// TIA Portal project "e199001v010" (V13)

(* hardware
DEVICE "Panel de operador_1"  KP900 Comfort
   slot 0: "HMI"  HMI  6AV2 124-1JC01-0AX0  13.0.1.0
   slot 1: "HMI_RT_1"  KP900 Comfort  6AV2 124-1JC01-0AX0  13.0.1.0
   slot 5: "Panel de operador_1.IE_CP_1"  Interfaz PROFINET
      slot 1: "Interfaz PROFINET_1"  Interfaz PROFINET
         slot 1: "Port_1"  Port
         slot 2: "Port_2"  Port
   slot 7: "Panel de operador_1.MPI/DP_CP_1"  Interfaz MPI/DP
*)

(* ===== HMI "HMI_RT_1" =====
connection "315_2DP": IF1 B, SIMATIC S7 300/400 MPI

HMI tags "Tabla de variables estándar"
   "Attendere1" : Byte, 1 s
   "LaserX" : Real, 1 s
   "TimeHBl" : S5Time, 1 s
   "SvoBobMin4" : Int, 1 s
   "PTMUX_MUXVAR_49" : Int, internal
   "Diam_filo10" : Real, 1 s
   "Color07" : Byte, 1 s
   "S_Int_1" : Int, 1 s
   "A_S_on07" : Bool, 1 s
   "TotalBlocks" : Int, 1 s
   "Diam_filo11" : Real, 1 s
   "Passo15" : Byte, 1 s
   "P14_Torque" : Int, 1 s
   "Trasf_Tipe" : Int, 1 s
   "DiamOutSvo" : Real, 1 s
   "CoefMul02" : Real, 1 s
   "PSvo_Current" : Int, 1 s
   "VelCin11" : Int, 1 s
   "R_F_Cur16" : Int, 1 s
   "P09_Power" : Int, 1 s
   "Q_elev" : Int, 1 s
   "RampJogDw" : Int, 1 s
   "RidMin14" : Int, 1 s
   "R_F_On07" : Bool, 1 s
   "TimLeft" : Real, 1 s
   "PTMUX_MUXVAR_45" : Int, internal
   "Q_bob_2" : Int, 1 s
   "P08_TempDriv" : Int, 1 s
   "VelMinChief" : Int, 1 s
   "P02_Speed" : Int, 1 s
   "Color05" : Byte, 1 s
   "Diam_filo14" : Real, 1 s
   "R_F_Cur01" : Int, 1 s
   "CoefMul03" : Real, 1 s
   "Mem_Rall" : Bool, 1 s
   "WearDieDw09" : Real, 1 s
   "P05_Current" : Int, 1 s
   "PTMUX_MUXVAR_46" : Int, internal
   "PTMUX_MUXVAR_37" : Int, internal
   "P07_Current" : Int, 1 s
   "R_F_On14" : Bool, 1 s
   "P06_Speed" : Int, 1 s
   "kW" : DInt, 1 s
   "Perc_WearAll" : Real, 1 s
   "Rall_manual" : Real, 1 s
   "SBPM_AGV_05" : Int, 1 s
   "Diam_filo04" : Real, 1 s
   "Ridu_12" : Int, 1 s
   "WearDieUp04" : Real, 1 s
   "WearDieDw14" : Real, 1 s
   "R_F_Cur06" : Int, 1 s
   "PTMUX_MUXVAR_10" : Int, internal
   "Check01" : Bool, 1 s
   "Gear5Elapsed" : Int, 1 s
   "Rst2" : Bool, 1 s
   "WearDieDw03" : Real, 1 s
   "AlTemQuad" : Int, 1 s
   "PJogL" : Int, 1 s
   "Diam_filo05" : Real, 1 s
   "RidMin10" : Int, 1 s
   "Color01" : Byte, 1 s
   "LaserOval" : Real, 1 s
   "PTMUX_MUXVAR_51" : Int, internal
   "RosetStat" : Byte, 1 s
   "WearDieDw04" : Real, 1 s
   "WearDieDw05" : Real, 1 s
   "P01_Speed" : Int, 1 s
   "P09_Current" : Int, 1 s
   "SBPM_AGV_12" : Int, 1 s
   "P05_Speed" : Int, 1 s
   "PBob_Power" : Int, 1 s
   "A_S_on05" : Bool, 1 s
   "Fil_rot_08" : Bool, 1 s
   "WearDieUp05" : Real, 1 s
   "Diam_filo02" : Real, 1 s
   "Passo11" : Byte, 1 s
   "PS_TempDrive" : Int, 1 s
   "P12_Torque" : Int, 1 s
   "Passo14" : Byte, 1 s
   "OTO_Actual" : Int, 1 s
   "Diam_Out" : Real, 1 s
   "Color09" : Byte, 1 s
   "OTO_Bargraph" : Int, 1 s
   "R_F_On15" : Bool, 1 s
   "P16_Current" : Int, 1 s
   "PTMUX_MUXVAR_26" : Int, internal
   "RidMin13" : Int, 1 s
   "Nr_recipe" : Int, 1 s
   "R_F_Cur15" : Int, 1 s
   "PTMUX_MUXVAR_53" : Int, internal
   "P13_Torque" : Int, 1 s
   "P12_Current" : Int, 1 s
   "PMat_Power" : Int, 1 s
   "P13_Current" : Int, 1 s
   "Matass" : Byte, 1 s
   "P16_Torque" : Int, 1 s
   "SvoBobMin2" : Int, 1 s
   "Color12" : Byte, 1 s
   "Fil_rot_01" : Bool, 1 s
   "PosizCarrell" : DInt, internal
   "SBPM_AGV_10" : Int, 1 s
   "BobMax1" : Int, 1 s
   "P15_Speed" : Int, 1 s
   "Ridu_06" : Int, 1 s
   "R_F_On10" : Bool, 1 s
   "WearDieUp09" : Real, 1 s
   "Acc_level" : Bool, 1 s
   "SvoBobMax1" : Int, 1 s
   "Diam_filo13" : Real, 1 s
   "D_Filt_Enc" : Int, 1 s
   "RidMin06" : Int, 1 s
   "Mux" : Int, 1 s
   "Fil_rot_09" : Bool, 1 s
   "PTMUX_MUXVAR_29" : Int, internal
   "VelMaxChief" : Int, 1 s
   "R_F_Cur14" : Int, 1 s
   "RidMin04" : Int, 1 s
   "SvoMax" : Int, 1 s
   "Counter_mat" : Real, 1 s
   "P15_Torque" : Int, 1 s
   "RidMin08" : Int, 1 s
   "PTMUX_MUXVAR_33" : Int, internal
   "CoefMul16" : Real, 1 s
   "P04_TempMot" : Int, 1 s
   "OTO_Min" : Int, 1 s
   "CoefMul09" : Real, 1 s
   "Gear4Elapsed" : Int, 1 s
   "P07_TempMot" : Int, 1 s
   "Ksensor" : Int, 1 s
   "CompAuto" : Bool, internal
   "Passo05" : Byte, 1 s
   "A_S_on01" : Bool, 1 s
   "P01_Torque" : Int, 1 s
   "Index" : Byte, 1 s
   "Tot_choic" : Byte, 1 s
   "WearDieUp12" : Real, 1 s
   "Fil_rot_10" : Bool, 1 s
   "Ridu_02" : Int, 1 s
   "Color08" : Byte, 1 s
   "RappDiam" : Int, 1 s   // E' il rapporto diametri bobine bobinatore
   "ControlSvo" : Bool, 1 s
   "DiamInSvo" : Real, 1 s
   "ControlStrat" : Bool, 1 s
   "Passo10" : Byte, 1 s
   "Laser2Thres" : Real, 1 s
   "SvoDiametro" : Int, 1 s
   "PTMUX_MUXVAR_25" : Int, internal
   "R_F_On03" : Bool, 1 s
   "Real_count" : Real, 1 s   // Metri parziali (prodotti)
   "Par_Type" : Byte, 1 s
   "TimeAccumulo" : Int, 1 s
   "P01_TempDriv" : Int, 1 s
   "Diam_filo06" : Real, 1 s
   "PSvo_Torque" : Int, 1 s
   "P10_Power" : Int, 1 s
   "VelCin14" : Int, 1 s
   "R_F_Cur12" : Int, 1 s
   "P15_Power" : Int, 1 s
   "Z_TIME" : WString[8], internal
   "GainCorr" : Int, 1 s
   "Diam_filo16" : Real, 1 s
   "RidMin16" : Int, 1 s
   "Pass_OTO" : Bool, 1 s   // Dichiarazione passo 1 se normale o OTO
   "CoefMul15" : Real, 1 s
   "PTMUX_MUXVAR_6" : Int, internal
   "Posizionam" : Int, internal
   "P03_TempMot" : Int, 1 s
   "WearDieDw02" : Real, 1 s
   "SBPM_AGV_04" : Int, 1 s
   "Passo06" : Byte, 1 s
   "PTMUX_MUXVAR_52" : Int, internal
   "P11_TempMot" : Int, 1 s
   "PTMUX_MUXVAR_1" : Int, internal
   "Elev_aut" : Bool, 1 s
   "Ridu_07" : Int, 1 s
   "Fil_rot_12" : Bool, 1 s
   "PTMUX_MUXVAR_7" : Int, internal
   "Param_Nr" : Int, 1 s
   "Passo02" : Byte, 1 s
   "VelCin08" : Int, 1 s
   "SBPM_AGV_15" : Int, 1 s
   "BobMin1" : Int, 1 s
   "Gear2Elapsed" : Int, 1 s
   "R_F_On02" : Bool, 1 s
   "Gear3Elapsed" : Int, 1 s
   "Diam_filo09" : Real, 1 s
   "P08_Speed" : Int, 1 s
   "R_F_On06" : Bool, 1 s
   "WearDieUp03" : Real, 1 s
   "SvoBobMin5" : Int, 1 s
   "SBPM_AGV_09" : Int, 1 s
   "Diam_filo03" : Real, 1 s
   "PTMUX_MUXVAR_8" : Int, internal
   "PTMUX_MUXVAR_16" : Int, internal
   "P13_Power" : Int, 1 s
   "Ridu_08" : Int, 1 s
   "PB_TempMot" : Int, 1 s
   "PTMUX_MUXVAR_27" : Int, internal
   "PT_Alarmas  1" : Array [0..19] of Int, 1 s
   "P07_Speed" : Int, 1 s
   "CoefMul10" : Real, 1 s
   "P11_TempDriv" : Int, 1 s
   "CoefMul07" : Real, 1 s
   "P13_TempMot" : Int, 1 s
   "Sfilaggio" : Bool, 1 s
   "P15_TempMot" : Int, 1 s
   "PTMUX_MUXVAR_36" : Int, internal
   "SBPM_AGV_16" : Int, 1 s
   "Ridu_16" : Int, 1 s
   "WearDieDw10" : Real, 1 s
   "VelCin06" : Int, 1 s
   "Gear4Set" : Int, 1 s
   "PMat_Torque" : Int, 1 s
   "VelCin03" : Int, 1 s
   "R_F_On11" : Bool, 1 s
   "DiamArrSvo" : Int, 1 s
   "Spool_choice" : Byte, 1 s
   "AGV_Set" : Bool, 1 s
   "R_F_Cur02" : Int, 1 s
   "CoefCorr" : Int, internal
   "WearDieUp14" : Real, 1 s
   "R_F_Cur08" : Int, 1 s
   "PMat_Speed" : Int, 1 s
   "LaserAlCh" : Bool, 1 s
   "PTMUX_MUXVAR_54" : Int, internal
   "Ridu_14" : Int, 1 s
   "Allineam" : Bool, 1 s
   "WearDieDw01" : Real, 1 s
   "Color04" : Byte, 1 s
   "Counter_traf" : Real, 1 s
   "PMat_Current" : Int, 1 s
   "PTMUX_MUXVAR_50" : Int, internal
   "OffAnalIn" : Int, 1 s
   "A_S_on16" : Bool, 1 s
   "PBobin" : Byte, 1 s
   "Diam_filo12" : Real, 1 s
   "VelMat" : Int, 1 s
   "PTMUX_MUXVAR_40" : Int, internal
   "PTMUX_MUXVAR_31" : Int, internal
   "SvoBobMax6" : Int, 1 s
   "Passo07" : Byte, 1 s
   "P09_TempDriv" : Int, 1 s
   "Pes_Specif" : Real, 1 s
   "Passo01" : Byte, 1 s
   "Ridu_01" : Int, 1 s
   "RappStrat3" : Int, 1 s
   "Fil_rot_05" : Bool, 1 s
   "P05_TempMot" : Int, 1 s
   "WearDieUp06" : Real, 1 s
   "WearDieUp11" : Real, 1 s
   "VelCin09" : Int, 1 s
   "P04_Torque" : Int, 1 s
   "P15_TempDriv" : Int, 1 s
   "PTMUX_MUXVAR_17" : Int, internal
   "Sirena" : Bool, 1 s
   "Perc_WearAvv" : Real, 1 s
   "PTMUX_MUXVAR_5" : Int, internal
   "PTMUX_MUXVAR_39" : Int, internal
   "PT_Acuses OP  2" : Array [0..4] of Word, 1 s
   "PTMUX_MUXVAR_47" : Int, internal
   "PTMUX_MUXVAR_24" : Int, internal
   "kg_total" : Real, 1 s
   "Gear5Set" : Int, 1 s
   "P07_Power" : Int, 1 s
   "JogDestra" : Int, internal
   "PTMUX_MUXVAR_38" : Int, internal
   "VelCin13" : Int, 1 s
   "P07_TempDriv" : Int, 1 s
   "Check05" : Bool, 1 s
   "P14_Power" : Int, 1 s
   "Ridu_10" : Int, 1 s
   "P09_Speed" : Int, 1 s
   "Fil_rot_11" : Bool, 1 s
   "Color13" : Byte, 1 s
   "BobTipo" : Bool, 1 s
   "Color03" : Byte, 1 s
   "Q_bob_3" : Int, 1 s
   "TimeForche" : S5Time, 1 s
   "Gear1Elapsed" : Int, 1 s
   "Imp_Exp" : Bool, 1 s
   "VelCin01" : Int, 1 s
   "PM_TempMot" : Int, 1 s
   "Rst1" : Bool, 1 s
   "Total" : Real, 1 s
   "PSvo_Power" : Int, 1 s
   "R_F_Cur09" : Int, 1 s
   "Stato_Linea" : Int, 1 s   // Visualizzazione stato linea
   "Q_bob_5" : Int, 1 s
   "Passo08" : Byte, 1 s
   "Vel_impostat" : Int, 1 s
   "CoefMul06" : Real, 1 s
   "P09_Torque" : Int, 1 s
   "PS_TempMot" : Int, 1 s
   "Gear1Set" : Int, 1 s
   "PTMUX_MUXVAR_35" : Int, internal
   "Exp_ImpQuest" : Bool, 1 s
   "SvoBobMin6" : Int, 1 s
   "Ridu_13" : Int, 1 s
   "SBPM" : Bool, 1 s   // Dichiarazione passo 1 se normale o OTO
   "RicFlangia" : Int, internal
   "A_S_on03" : Bool, 1 s
   "RidMin01" : Int, 1 s
   "OTO_BarUP" : Int, 1 s
   "Check02" : Bool, 1 s
   "TimeH2Fil" : S5Time, 1 s
   "PT_Acuses OP  1" : Array [0..9] of Int, 1 s
   "P11_Torque" : Int, 1 s
   "P14_TempDriv" : Int, 1 s
   "Life_hours" : DInt, 1 s
   "Ral_Aut_Cal" : Real, 1 s
   "JogSinistra" : Int, internal
   "P10_TempDriv" : Int, 1 s
   "PTMUX_MUXVAR_32" : Int, internal
   "A_S_on06" : Bool, 1 s
   "CoefMul05" : Real, 1 s
   "P03_Torque" : Int, 1 s
   "Fil_rot_03" : Bool, 1 s
   "P15_Current" : Int, 1 s
   "A_S_on14" : Bool, 1 s
   "SvoBobMin1" : Int, 1 s
   "RappStrat2" : Int, 1 s
   "P08_TempMot" : Int, 1 s
   "P03_Speed" : Int, 1 s
   "PTMUX_MUXVAR_34" : Int, internal
   "PTMUX_MUXVAR_30" : Int, internal
   "P14_Speed" : Int, 1 s
   "A_S_on12" : Bool, 1 s
   "Imp_count" : Real, 1 s   // Metri impostati
   "P04_TempDriv" : Int, 1 s
   "R_F_On09" : Bool, 1 s
   "JogStrat" : Int, 1 s
   "RappStrat1" : Int, 1 s
   "A_S_on13" : Bool, 1 s
   "Color02" : Byte, 1 s
   "SvoMin" : Int, 1 s
   "VelCin12" : Int, 1 s
   "RappStrat4" : Int, 1 s
   "K_Stratific" : Int, 1 s
   "BobMax2" : Int, 1 s
   "RidMin02" : Int, 1 s
   "P06_TempMot" : Int, 1 s
   "P05_Torque" : Int, 1 s
   "RidMin05" : Int, 1 s
   "SvoBobMax4" : Int, 1 s
   "OTO_MinRid" : Int, 1 s
   "Passo09" : Byte, 1 s
   "P02_Torque" : Int, 1 s
   "SistMisure" : Bool, 1 s
   "RosettVel" : Int, 1 s
   "PTMUX_MUXVAR_12" : Int, internal
   "BobCoppia" : Int, 1 s
   "SBPM_AGV_11" : Int, 1 s
   "CoefMul12" : Real, 1 s
   "PTMUX_MUXVAR_19" : Int, internal
   "Diam_filo01" : Real, 1 s
   "S_Int_5" : Int, 1 s
   "P02_Current" : Int, 1 s
   "MaxSens" : Int, 1 s
   "Block_Choice" : Int, 1 s
   "P10_Speed" : Int, 1 s
   "RidMin12" : Int, 1 s
   "R_F_Cur03" : Int, 1 s
   "R_F_Cur07" : Int, 1 s
   "PTMUX_MUXVAR_56" : Int, internal
   "Domanda" : Bool, 1 s
   "S_IntTime" : Int, 1 s
   "PTMUX_MUXVAR_41" : Int, internal
   "Ridu_09" : Int, 1 s
   "VelCin15" : Int, 1 s
   "A_S_on02" : Bool, 1 s
   "Ridu_11" : Int, 1 s
   "P16_Speed" : Int, 1 s
   "CoefMul04" : Real, 1 s
   "PTMUX_MUXVAR_2" : Int, internal
   "P07_Torque" : Int, 1 s
   "Color11" : Byte, 1 s
   "P04_Current" : Int, 1 s
   "Passo04" : Byte, 1 s
   "LaserY" : Real, 1 s
   "LaserMedio" : Real, 1 s
   "kg" : Bool, internal
   "WearDieUp01" : Real, 1 s
   "R_F_Cur05" : Int, 1 s
   "Ridu_15" : Int, 1 s
   "Diam_filo08" : Real, 1 s
   "P12_Speed" : Int, 1 s
   "Contametri" : Byte, 1 s
   "PBob_Speed" : Int, 1 s
   "WearDieUp07" : Real, 1 s
   "SBPM_AGV_03" : Int, 1 s
   "VelCin02" : Int, 1 s
   "RidMin11" : Int, 1 s
   "BobMin2" : Int, 1 s
   "Sens_Gain" : Int, 1 s
   "PTMUX_MUXVAR_22" : Int, internal
   "Color14" : Byte, 1 s
   "A_S_on11" : Bool, 1 s
   "InvSinistra" : Int, internal
   "P08_Torque" : Int, 1 s
   "PTMUX_MUXVAR_57" : Int, internal
   "Rst4" : Bool, 1 s
   "R_F_Cur10" : Int, 1 s
   "Color16" : Byte, 1 s
   "PBob_Torque" : Int, 1 s
   "PTMUX_MUXVAR_23" : Int, internal
   "P08_Current" : Int, 1 s
   "PTMUX_MUXVAR_11" : Int, internal
   "P02_TempMot" : Int, 1 s
   "Svolgitore" : Byte, 1 s
   "Gear2Set" : Int, 1 s
   "P02_TempDriv" : Int, 1 s
   "SBPM_AGV_07" : Int, 1 s
   "Elevator" : Bool, 1 s
   "A_S_on10" : Bool, 1 s
   "VelCin10" : Int, 1 s
   "PT_Alarmas  2" : Array [0..9] of Word, 1 s
   "CoefMul11" : Real, 1 s
   "Color10" : Byte, 1 s
   "Rst3" : Bool, 1 s
   "P03_Power" : Int, 1 s
   "R_F_On08" : Bool, 1 s
   "SvoBobMax3" : Int, 1 s
   "P10_TempMot" : Int, 1 s
   "PTMUX_MUXVAR_44" : Int, internal
   "WearDieUp10" : Real, 1 s
   "PAct_Sen" : Int, 1 s
   "Sel_count" : Bool, 1 s
   "Diam_filo07" : Real, 1 s
   "R_F_On13" : Bool, 1 s
   "Fil_rot_06" : Bool, 1 s
   "PTMUX_MUXVAR_43" : Int, internal
   "CoefMul14" : Real, 1 s
   "Fil_rot_04" : Bool, 1 s
   "Fast_Dw" : Int, 1 s
   "PTMUX_MUXVAR_20" : Int, internal
   "PTMUX_MUXVAR_15" : Int, internal
   "Svo_Spools" : Byte, 1 s
   "SvoBobMax2" : Int, 1 s
   "kg_parz" : Real, 1 s
   "Attendere" : Bool, 1 s
   "R_F_Cur04" : Int, 1 s
   "AGV" : DInt, 1 s
   "T_Rosett" : Int, internal
   "R_F_Cur13" : Int, 1 s
   "P04_Speed" : Int, 1 s
   "PJogV" : Int, 1 s
   "Fil_rot_07" : Bool, 1 s
   "BobTirVel" : Bool, 1 s
   "S_Rosett" : Int, internal
   "PTMUX_MUXVAR_14" : Int, internal
   "VelCin16" : Int, 1 s
   "PTMUX_MUXVAR_18" : Int, internal
   "Ridu_04" : Int, 1 s
   "Real_Sens" : Int, 1 s
   "PTMUX_MUXVAR_55" : Int, internal
   "Color06" : Byte, 1 s
   "Q_bob_6" : Int, 1 s
   "OTOMotorized" : Bool, 1 s   // Dichiarazione passo 1 motorizzato o no
   "RidMin07" : Int, 1 s
   "Passo16" : Byte, 1 s
   "Gear3Set" : Int, 1 s
   "RampJogUp" : Int, 1 s
   "WearDieDw07" : Real, 1 s
   "P06_Current" : Int, 1 s
   "SvoBobMin3" : Int, 1 s
   "PTMUX_MUXVAR_28" : Int, internal
   "Diam_filoM" : Real, 1 s
   "Passo12" : Byte, 1 s
   "SBPM_AGV_01" : Int, 1 s
   "WearDieUp13" : Real, 1 s
   "Rosett" : Bool, 1 s
   "Fil_rot_14" : Bool, 1 s
   "Attendere3" : Byte, 1 s
   "WearDieDw06" : Real, 1 s
   "R_F_On16" : Bool, 1 s
   "P16_TempMot" : Int, 1 s
   "WearDieDw12" : Real, 1 s
   "Passo13" : Byte, 1 s
   "RidMin03" : Int, 1 s
   "PTMUX_MUXVAR_9" : Int, internal
   "Diam_filo15" : Real, 1 s
   "P08_Power" : Int, 1 s
   "LaserChoic" : Bool, 1 s
   "P16_Power" : Int, 1 s
   "OTO_Imposed" : Int, 1 s
   "WearDieUp08" : Real, 1 s
   "DiamManual" : Real, 1 s
   "A_S_on09" : Bool, 1 s
   "PT_Imagen de los LED  1" : Array [0..3] of Int, 1 s
   "CoefMul01" : Real, 1 s
   "P09_TempMot" : Int, 1 s
   "Check03" : Bool, 1 s
   "Task_Id" : Int, 1 s
   "OTO_Rid" : Int, 1 s
   "P02_Power" : Int, 1 s
   "DistanzaPx" : DInt, internal
   "LaserStato" : Int, 1 s
   "Recipe_Wait" : Int, 1 s
   "OutChoice" : Byte, 1 s
   "A_S_on08" : Bool, 1 s
   "P06_Power" : Int, 1 s
   "Ridu_03" : Int, 1 s
   "TempQuad" : Int, 1 s
   "R_F_On01" : Bool, 1 s
   "PTMUX_MUXVAR_42" : Int, internal
   "P11_Current" : Int, 1 s
   "PTMUX_MUXVAR_3" : Int, internal
   "S_Int_4" : Int, 1 s
   "VelRal" : Int, 1 s
   "R_F_Cur11" : Int, 1 s
   "Color15" : Byte, 1 s
   "Worked_hours" : DInt, 1 s
   "OTO_Max" : Int, 1 s
   "P06_Torque" : Int, 1 s
   "kg_imp" : Real, 1 s
   "A_S_on04" : Bool, 1 s
   "AnticipoSvo" : Int, 1 s
   "D_Prop_1" : Int, 1 s
   "VelSfilag" : Int, 1 s
   "Slow_Up" : Int, 1 s
   "R_F_On12" : Bool, 1 s
   "PTMUX_MUXVAR_13" : Int, internal
   "Fil_rot_16" : Bool, 1 s
   "P04_Power" : Int, 1 s
   "PTMUX_MUXVAR_4" : Int, internal
   "SBPM_AGV_14" : Int, 1 s
   "RealSpINT" : Int, 1 s   // Velocita' m/s in REAL
   "WearDieUp02" : Real, 1 s
   "P03_Current" : Int, 1 s
   "WearDieDw11" : Real, 1 s
   "P10_Torque" : Int, 1 s
   "WearDieDw08" : Real, 1 s
   "OTO_BarDW" : Int, 1 s
   "P12_TempDriv" : Int, 1 s
   "R_F_On05" : Bool, 1 s
   "Rst5" : Bool, 1 s
   "VelCin07" : Int, 1 s
   "Attesa2" : Bool, 1 s
   "PSvo_Speed" : Int, 1 s
   "P14_Current" : Int, 1 s
   "S_Int_2" : Int, 1 s
   "S_Prop_2" : Int, 1 s
   "P12_Power" : Int, 1 s
   "Passo03" : Byte, 1 s
   "P13_TempDriv" : Int, 1 s
   "Laser1Thres" : Real, 1 s
   "Attesa1" : Bool, 1 s
   "CoefMul13" : Real, 1 s
   "Fil_rot_15" : Bool, 1 s
   "P01_Power" : Int, 1 s
   "SBPM_AGV_02" : Int, 1 s
   "D_Int" : Int, 1 s
   "Z_DATE" : WString[10], internal
   "CoefMul08" : Real, 1 s
   "Check04" : Bool, 1 s
   "PTMUX_MUXVAR_21" : Int, internal
   "P12_TempMot" : Int, 1 s
   "ON_SS" : Byte, 1 s
   "SBPM_AGV_13" : Int, 1 s
   "P10_Current" : Int, 1 s
   "MinSens" : Int, 1 s
   "Q_bob_1" : Int, 1 s
   "Slow_dw" : Int, 1 s
   "Max_vel" : Int, 1 s
   "SBPM_AGV_08" : Int, 1 s
   "S_Prop_1" : Int, 1 s
   "Fil_rot_13" : Bool, 1 s
   "BypassDati" : Bool, 1 s
   "PM_TempDriv" : Int, 1 s
   "P13_Speed" : Int, 1 s
   "Reset_kW" : Bool, 1 s
   "P01_Current" : Int, 1 s
   "A_S_on15" : Bool, 1 s
   "PB_TempDrive" : Int, 1 s
   "Q_bob_4" : Int, 1 s
   "BobTiro" : Int, 1 s
   "TimeVenBloc" : S5Time, 1 s
   "PTMUX_MUXVAR_48" : Int, internal
   "P11_Power" : Int, 1 s
   "Die_Wear_Ch" : Byte, 1 s
   "D_Prop_2" : Int, 1 s
   "P16_TempDriv" : Int, 1 s
   "WearDieDw13" : Real, 1 s
   "Value" : DInt, 1 s
   "SvoBobMax5" : Int, 1 s
   "RidMin15" : Int, 1 s
   "ColorSvolg" : Byte, 1 s
   "Ridu_05" : Int, 1 s
   "PT_Avisos de servicio  1" : Array [0..4] of Int, 1 s
   "R_F_On04" : Bool, 1 s
   "P03_TempDriv" : Int, 1 s
   "VelCin05" : Int, 1 s
   "P11_Speed" : Int, 1 s
   "SBPM_AGV_06" : Int, 1 s
   "Mux1" : Int, 1 s
   "VelCin04" : Int, 1 s
   "PBob_Current" : Int, 1 s
   "InvDestra" : Int, internal
   "P14_TempMot" : Int, 1 s
   "P06_TempDriv" : Int, 1 s
   "P01_TempMot" : Int, 1 s
   "Min_vel" : Int, 1 s
   "P05_TempDriv" : Int, 1 s
   "TimeStratCal" : Int, 1 s
   "P05_Power" : Int, 1 s
   "BobDiametro" : Int, 1 s
   "Sens_Deriv" : Int, 1 s
   "Pilota" : Int, 1 s
   "Fil_rot_02" : Bool, 1 s
   "Time_1" : DateTime, internal

discrete alarms
   43: '', class Warnings, trigger "PT_Avisos de servicio  1" bit 42
   2018: '', class Errors, trigger "PT_Acuses OP  1" bit 17
   2209: '', class Errors, trigger "PT_Acuses OP  2" bit 48
   2034: '', class Errors, trigger "PT_Acuses OP  1" bit 33
   17: '', class Warnings, trigger "PT_Avisos de servicio  1" bit 16
   2: '', class Warnings, trigger "PT_Avisos de servicio  1" bit 1
   2189: '', class Errors, trigger "PT_Acuses OP  2" bit 28
   2129: '', class Errors, trigger "PT_Acuses OP  1" bit 128
   2019: '', class Errors, trigger "PT_Acuses OP  1" bit 18
   2098: '', class Errors, trigger "PT_Acuses OP  1" bit 97
   2072: '', class Errors, trigger "PT_Acuses OP  1" bit 71
   24: '', class Warnings, trigger "PT_Avisos de servicio  1" bit 23
   2188: '', class Errors, trigger "PT_Acuses OP  2" bit 27
   2181: '', class Errors, trigger "PT_Acuses OP  2" bit 20
   2014: '', class Errors, trigger "PT_Acuses OP  1" bit 13
   2049: '', class Errors, trigger "PT_Acuses OP  1" bit 48
   2141: '', class Errors, trigger "PT_Acuses OP  1" bit 140
   10: '', class Warnings, trigger "PT_Avisos de servicio  1" bit 9
   2023: '', class Errors, trigger "PT_Acuses OP  1" bit 22
   2031: '', class Errors, trigger "PT_Acuses OP  1" bit 30
   2219: '', class Errors, trigger "PT_Acuses OP  2" bit 58
   2200: '', class Errors, trigger "PT_Acuses OP  2" bit 39
   40: '', class Warnings, trigger "PT_Avisos de servicio  1" bit 39
   2193: '', class Errors, trigger "PT_Acuses OP  2" bit 32
   2128: '', class Errors, trigger "PT_Acuses OP  1" bit 127
   2140: '', class Errors, trigger "PT_Acuses OP  1" bit 139
   2053: '', class Errors, trigger "PT_Acuses OP  1" bit 52
   70: '', class Warnings, trigger "PT_Avisos de servicio  1" bit 69
   2061: '', class Errors, trigger "PT_Acuses OP  1" bit 60
   2135: '', class Errors, trigger "PT_Acuses OP  1" bit 134
   2126: '', class Errors, trigger "PT_Acuses OP  1" bit 125
   2065: '', class Errors, trigger "PT_Acuses OP  1" bit 64
   2206: '', class Errors, trigger "PT_Acuses OP  2" bit 45
   73: '', class Warnings, trigger "PT_Avisos de servicio  1" bit 72
   2199: '', class Errors, trigger "PT_Acuses OP  2" bit 38
   71: '', class Warnings, trigger "PT_Avisos de servicio  1" bit 70
   2158: '', class Errors, trigger "PT_Acuses OP  1" bit 157
   2038: '', class Errors, trigger "PT_Acuses OP  1" bit 37
   19: '', class Warnings, trigger "PT_Avisos de servicio  1" bit 18
   2081: '', class Errors, trigger "PT_Acuses OP  1" bit 80
   37: '', class Warnings, trigger "PT_Avisos de servicio  1" bit 36
   3: '', class Warnings, trigger "PT_Avisos de servicio  1" bit 2
   2238: '', class Errors, trigger "PT_Acuses OP  2" bit 77
   2201: '', class Errors, trigger "PT_Acuses OP  2" bit 40
   2008: '', class Errors, trigger "PT_Acuses OP  1" bit 7
   2032: '', class Errors, trigger "PT_Acuses OP  1" bit 31
   2145: '', class Errors, trigger "PT_Acuses OP  1" bit 144
   2143: '', class Errors, trigger "PT_Acuses OP  1" bit 142
   2134: '', class Errors, trigger "PT_Acuses OP  1" bit 133
   2056: '', class Errors, trigger "PT_Acuses OP  1" bit 55
   2004: '', class Errors, trigger "PT_Acuses OP  1" bit 3
   2043: '', class Errors, trigger "PT_Acuses OP  1" bit 42
   2216: '', class Errors, trigger "PT_Acuses OP  2" bit 55
   2234: '', class Errors, trigger "PT_Acuses OP  2" bit 73
   27: '', class Warnings, trigger "PT_Avisos de servicio  1" bit 26
   2133: '', class Errors, trigger "PT_Acuses OP  1" bit 132
   2113: '', class Errors, trigger "PT_Acuses OP  1" bit 112
   31: '', class Warnings, trigger "PT_Avisos de servicio  1" bit 30
   2170: '', class Errors, trigger "PT_Acuses OP  2" bit 9
   2162: '', class Errors, trigger "PT_Acuses OP  2" bit 1
   29: '', class Warnings, trigger "PT_Avisos de servicio  1" bit 28
   2187: '', class Errors, trigger "PT_Acuses OP  2" bit 26
   2094: '', class Errors, trigger "PT_Acuses OP  1" bit 93
   2041: '', class Errors, trigger "PT_Acuses OP  1" bit 40
   2076: '', class Errors, trigger "PT_Acuses OP  1" bit 75
   2084: '', class Errors, trigger "PT_Acuses OP  1" bit 83
   2215: '', class Errors, trigger "PT_Acuses OP  2" bit 54
   2131: '', class Errors, trigger "PT_Acuses OP  1" bit 130
   2195: '', class Errors, trigger "PT_Acuses OP  2" bit 34
   2205: '', class Errors, trigger "PT_Acuses OP  2" bit 44
   78: '', class Warnings, trigger "PT_Avisos de servicio  1" bit 77
   2079: '', class Errors, trigger "PT_Acuses OP  1" bit 78
   2068: '', class Errors, trigger "PT_Acuses OP  1" bit 67
   2196: '', class Errors, trigger "PT_Acuses OP  2" bit 35
   2123: '', class Errors, trigger "PT_Acuses OP  1" bit 122
   2152: '', class Errors, trigger "PT_Acuses OP  1" bit 151
   2112: '', class Errors, trigger "PT_Acuses OP  1" bit 111
   2211: '', class Errors, trigger "PT_Acuses OP  2" bit 50
   2077: '', class Errors, trigger "PT_Acuses OP  1" bit 76
   46: '', class Warnings, trigger "PT_Avisos de servicio  1" bit 45
   77: '', class Warnings, trigger "PT_Avisos de servicio  1" bit 76
   33: '', class Warnings, trigger "PT_Avisos de servicio  1" bit 32
   2148: '', class Errors, trigger "PT_Acuses OP  1" bit 147
   2064: '', class Errors, trigger "PT_Acuses OP  1" bit 63
   65: '', class Warnings, trigger "PT_Avisos de servicio  1" bit 64
   2237: '', class Errors, trigger "PT_Acuses OP  2" bit 76
   79: '', class Warnings, trigger "PT_Avisos de servicio  1" bit 78
   2218: '', class Errors, trigger "PT_Acuses OP  2" bit 57
   2075: '', class Errors, trigger "PT_Acuses OP  1" bit 74
   2167: '', class Errors, trigger "PT_Acuses OP  2" bit 6
   2073: '', class Errors, trigger "PT_Acuses OP  1" bit 72
   2225: '', class Errors, trigger "PT_Acuses OP  2" bit 64
   2070: '', class Errors, trigger "PT_Acuses OP  1" bit 69
   2222: '', class Errors, trigger "PT_Acuses OP  2" bit 61
   22: '', class Warnings, trigger "PT_Avisos de servicio  1" bit 21
   2092: '', class Errors, trigger "PT_Acuses OP  1" bit 91
   2208: '', class Errors, trigger "PT_Acuses OP  2" bit 47
   56: '', class Warnings, trigger "PT_Avisos de servicio  1" bit 55
   6: '', class Warnings, trigger "PT_Avisos de servicio  1" bit 5
   25: '', class Warnings, trigger "PT_Avisos de servicio  1" bit 24
   2045: '', class Errors, trigger "PT_Acuses OP  1" bit 44
   2161: '', class Errors, trigger "PT_Acuses OP  2" bit 0
   2122: '', class Errors, trigger "PT_Acuses OP  1" bit 121
   2192: '', class Errors, trigger "PT_Acuses OP  2" bit 31
   2108: '', class Errors, trigger "PT_Acuses OP  1" bit 107
   2011: '', class Errors, trigger "PT_Acuses OP  1" bit 10
   2230: '', class Errors, trigger "PT_Acuses OP  2" bit 69
   2052: '', class Errors, trigger "PT_Acuses OP  1" bit 51
   2163: '', class Errors, trigger "PT_Acuses OP  2" bit 2
   2027: '', class Errors, trigger "PT_Acuses OP  1" bit 26
   2093: '', class Errors, trigger "PT_Acuses OP  1" bit 92
   2026: '', class Errors, trigger "PT_Acuses OP  1" bit 25
   68: '', class Warnings, trigger "PT_Avisos de servicio  1" bit 67
   2144: '', class Errors, trigger "PT_Acuses OP  1" bit 143
   2150: '', class Errors, trigger "PT_Acuses OP  1" bit 149
   2005: '', class Errors, trigger "PT_Acuses OP  1" bit 4
   2036: '', class Errors, trigger "PT_Acuses OP  1" bit 35
   72: '', class Warnings, trigger "PT_Avisos de servicio  1" bit 71
   2040: '', class Errors, trigger "PT_Acuses OP  1" bit 39
   48: '', class Warnings, trigger "PT_Avisos de servicio  1" bit 47
   2146: '', class Errors, trigger "PT_Acuses OP  1" bit 145
   2042: '', class Errors, trigger "PT_Acuses OP  1" bit 41
   55: '', class Warnings, trigger "PT_Avisos de servicio  1" bit 54
   2174: '', class Errors, trigger "PT_Acuses OP  2" bit 13
   2210: '', class Errors, trigger "PT_Acuses OP  2" bit 49
   2235: '', class Errors, trigger "PT_Acuses OP  2" bit 74
   5: '', class Warnings, trigger "PT_Avisos de servicio  1" bit 4
   57: '', class Warnings, trigger "PT_Avisos de servicio  1" bit 56
   74: '', class Warnings, trigger "PT_Avisos de servicio  1" bit 73
   2137: '', class Errors, trigger "PT_Acuses OP  1" bit 136
   2138: '', class Errors, trigger "PT_Acuses OP  1" bit 137
   80: '', class Warnings, trigger "PT_Avisos de servicio  1" bit 79
   2062: '', class Errors, trigger "PT_Acuses OP  1" bit 61
   8: '', class Warnings, trigger "PT_Avisos de servicio  1" bit 7
   2178: '', class Errors, trigger "PT_Acuses OP  2" bit 17
   11: '', class Warnings, trigger "PT_Avisos de servicio  1" bit 10
   2217: '', class Errors, trigger "PT_Acuses OP  2" bit 56
   13: '', class Warnings, trigger "PT_Avisos de servicio  1" bit 12
   2149: '', class Errors, trigger "PT_Acuses OP  1" bit 148
   2120: '', class Errors, trigger "PT_Acuses OP  1" bit 119
   2213: '', class Errors, trigger "PT_Acuses OP  2" bit 52
   2207: '', class Errors, trigger "PT_Acuses OP  2" bit 46
   2071: '', class Errors, trigger "PT_Acuses OP  1" bit 70
   2033: '', class Errors, trigger "PT_Acuses OP  1" bit 32
   2059: '', class Errors, trigger "PT_Acuses OP  1" bit 58
   2088: '', class Errors, trigger "PT_Acuses OP  1" bit 87
   2010: '', class Errors, trigger "PT_Acuses OP  1" bit 9
   2156: '', class Errors, trigger "PT_Acuses OP  1" bit 155
   2022: '', class Errors, trigger "PT_Acuses OP  1" bit 21
   7: '', class Warnings, trigger "PT_Avisos de servicio  1" bit 6
   2047: '', class Errors, trigger "PT_Acuses OP  1" bit 46
   2090: '', class Errors, trigger "PT_Acuses OP  1" bit 89
   2074: '', class Errors, trigger "PT_Acuses OP  1" bit 73
   15: '', class Warnings, trigger "PT_Avisos de servicio  1" bit 14
   4: '', class Warnings, trigger "PT_Avisos de servicio  1" bit 3
   2025: '', class Errors, trigger "PT_Acuses OP  1" bit 24
   75: '', class Warnings, trigger "PT_Avisos de servicio  1" bit 74
   61: '', class Warnings, trigger "PT_Avisos de servicio  1" bit 60
   2114: '', class Errors, trigger "PT_Acuses OP  1" bit 113
   2091: '', class Errors, trigger "PT_Acuses OP  1" bit 90
   2117: '', class Errors, trigger "PT_Acuses OP  1" bit 116
   21: '', class Warnings, trigger "PT_Avisos de servicio  1" bit 20
   49: '', class Warnings, trigger "PT_Avisos de servicio  1" bit 48
   2153: '', class Errors, trigger "PT_Acuses OP  1" bit 152
   50: '', class Warnings, trigger "PT_Avisos de servicio  1" bit 49
   32: '', class Warnings, trigger "PT_Avisos de servicio  1" bit 31
   2030: '', class Errors, trigger "PT_Acuses OP  1" bit 29
   2085: '', class Errors, trigger "PT_Acuses OP  1" bit 84
   2116: '', class Errors, trigger "PT_Acuses OP  1" bit 115
   2173: '', class Errors, trigger "PT_Acuses OP  2" bit 12
   2194: '', class Errors, trigger "PT_Acuses OP  2" bit 33
   2080: '', class Errors, trigger "PT_Acuses OP  1" bit 79
   2009: '', class Errors, trigger "PT_Acuses OP  1" bit 8
   16: '', class Warnings, trigger "PT_Avisos de servicio  1" bit 15
   2055: '', class Errors, trigger "PT_Acuses OP  1" bit 54
   2078: '', class Errors, trigger "PT_Acuses OP  1" bit 77
   2159: '', class Errors, trigger "PT_Acuses OP  1" bit 158
   76: '', class Warnings, trigger "PT_Avisos de servicio  1" bit 75
   2171: '', class Errors, trigger "PT_Acuses OP  2" bit 10
   2233: '', class Errors, trigger "PT_Acuses OP  2" bit 72
   2035: '', class Errors, trigger "PT_Acuses OP  1" bit 34
   2104: '', class Errors, trigger "PT_Acuses OP  1" bit 103
   2226: '', class Errors, trigger "PT_Acuses OP  2" bit 65
   2186: '', class Errors, trigger "PT_Acuses OP  2" bit 25
   2115: '', class Errors, trigger "PT_Acuses OP  1" bit 114
   2125: '', class Errors, trigger "PT_Acuses OP  1" bit 124
   2050: '', class Errors, trigger "PT_Acuses OP  1" bit 49
   45: '', class Warnings, trigger "PT_Avisos de servicio  1" bit 44
   2157: '', class Errors, trigger "PT_Acuses OP  1" bit 156
   2086: '', class Errors, trigger "PT_Acuses OP  1" bit 85
   2087: '', class Errors, trigger "PT_Acuses OP  1" bit 86
   2111: '', class Errors, trigger "PT_Acuses OP  1" bit 110
   2183: '', class Errors, trigger "PT_Acuses OP  2" bit 22
   2180: '', class Errors, trigger "PT_Acuses OP  2" bit 19
   2166: '', class Errors, trigger "PT_Acuses OP  2" bit 5
   2048: '', class Errors, trigger "PT_Acuses OP  1" bit 47
   2142: '', class Errors, trigger "PT_Acuses OP  1" bit 141
   58: '', class Warnings, trigger "PT_Avisos de servicio  1" bit 57
   2101: '', class Errors, trigger "PT_Acuses OP  1" bit 100
   9: '', class Warnings, trigger "PT_Avisos de servicio  1" bit 8
   2185: '', class Errors, trigger "PT_Acuses OP  2" bit 24
   2229: '', class Errors, trigger "PT_Acuses OP  2" bit 68
   1: '', class Warnings, trigger "PT_Avisos de servicio  1" bit 0
   2154: '', class Errors, trigger "PT_Acuses OP  1" bit 153
   2082: '', class Errors, trigger "PT_Acuses OP  1" bit 81
   2124: '', class Errors, trigger "PT_Acuses OP  1" bit 123
   2103: '', class Errors, trigger "PT_Acuses OP  1" bit 102
   2169: '', class Errors, trigger "PT_Acuses OP  2" bit 8
   2236: '', class Errors, trigger "PT_Acuses OP  2" bit 75
   2164: '', class Errors, trigger "PT_Acuses OP  2" bit 3
   2118: '', class Errors, trigger "PT_Acuses OP  1" bit 117
   2106: '', class Errors, trigger "PT_Acuses OP  1" bit 105
   2139: '', class Errors, trigger "PT_Acuses OP  1" bit 138
   2202: '', class Errors, trigger "PT_Acuses OP  2" bit 41
   39: '', class Warnings, trigger "PT_Avisos de servicio  1" bit 38
   67: '', class Warnings, trigger "PT_Avisos de servicio  1" bit 66
   2107: '', class Errors, trigger "PT_Acuses OP  1" bit 106
   2231: '', class Errors, trigger "PT_Acuses OP  2" bit 70
   2024: '', class Errors, trigger "PT_Acuses OP  1" bit 23
   2177: '', class Errors, trigger "PT_Acuses OP  2" bit 16
   2190: '', class Errors, trigger "PT_Acuses OP  2" bit 29
   2083: '', class Errors, trigger "PT_Acuses OP  1" bit 82
   2096: '', class Errors, trigger "PT_Acuses OP  1" bit 95
   2203: '', class Errors, trigger "PT_Acuses OP  2" bit 42
   2046: '', class Errors, trigger "PT_Acuses OP  1" bit 45
   2184: '', class Errors, trigger "PT_Acuses OP  2" bit 23
   12: '', class Warnings, trigger "PT_Avisos de servicio  1" bit 11
   2069: '', class Errors, trigger "PT_Acuses OP  1" bit 68
   2109: '', class Errors, trigger "PT_Acuses OP  1" bit 108
   2176: '', class Errors, trigger "PT_Acuses OP  2" bit 15
   2021: '', class Errors, trigger "PT_Acuses OP  1" bit 20
   2220: '', class Errors, trigger "PT_Acuses OP  2" bit 59
   2165: '', class Errors, trigger "PT_Acuses OP  2" bit 4
   2121: '', class Errors, trigger "PT_Acuses OP  1" bit 120
   52: '', class Warnings, trigger "PT_Avisos de servicio  1" bit 51
   34: '', class Warnings, trigger "PT_Avisos de servicio  1" bit 33
   2110: '', class Errors, trigger "PT_Acuses OP  1" bit 109
   2221: '', class Errors, trigger "PT_Acuses OP  2" bit 60
   51: '', class Warnings, trigger "PT_Avisos de servicio  1" bit 50
   2058: '', class Errors, trigger "PT_Acuses OP  1" bit 57
   53: '', class Warnings, trigger "PT_Avisos de servicio  1" bit 52
   2204: '', class Errors, trigger "PT_Acuses OP  2" bit 43
   2063: '', class Errors, trigger "PT_Acuses OP  1" bit 62
   2003: '', class Errors, trigger "PT_Acuses OP  1" bit 2
   2130: '', class Errors, trigger "PT_Acuses OP  1" bit 129
   2037: '', class Errors, trigger "PT_Acuses OP  1" bit 36
   2160: '', class Errors, trigger "PT_Acuses OP  1" bit 159
   62: '', class Warnings, trigger "PT_Avisos de servicio  1" bit 61
   69: '', class Warnings, trigger "PT_Avisos de servicio  1" bit 68
   2097: '', class Errors, trigger "PT_Acuses OP  1" bit 96
   35: '', class Warnings, trigger "PT_Avisos de servicio  1" bit 34
   44: '', class Warnings, trigger "PT_Avisos de servicio  1" bit 43
   20: '', class Warnings, trigger "PT_Avisos de servicio  1" bit 19
   2099: '', class Errors, trigger "PT_Acuses OP  1" bit 98
   30: '', class Warnings, trigger "PT_Avisos de servicio  1" bit 29
   2057: '', class Errors, trigger "PT_Acuses OP  1" bit 56
   2102: '', class Errors, trigger "PT_Acuses OP  1" bit 101
   2095: '', class Errors, trigger "PT_Acuses OP  1" bit 94
   2039: '', class Errors, trigger "PT_Acuses OP  1" bit 38
   2017: '', class Errors, trigger "PT_Acuses OP  1" bit 16
   38: '', class Warnings, trigger "PT_Avisos de servicio  1" bit 37
   2191: '', class Errors, trigger "PT_Acuses OP  2" bit 30
   2001: '', class Errors, trigger "PT_Acuses OP  1" bit 0
   2168: '', class Errors, trigger "PT_Acuses OP  2" bit 7
   63: '', class Warnings, trigger "PT_Avisos de servicio  1" bit 62
   2044: '', class Errors, trigger "PT_Acuses OP  1" bit 43
   2227: '', class Errors, trigger "PT_Acuses OP  2" bit 66
   2105: '', class Errors, trigger "PT_Acuses OP  1" bit 104
   2175: '', class Errors, trigger "PT_Acuses OP  2" bit 14
   2198: '', class Errors, trigger "PT_Acuses OP  2" bit 37
   60: '', class Warnings, trigger "PT_Avisos de servicio  1" bit 59
   2067: '', class Errors, trigger "PT_Acuses OP  1" bit 66
   2089: '', class Errors, trigger "PT_Acuses OP  1" bit 88
   2015: '', class Errors, trigger "PT_Acuses OP  1" bit 14
   41: '', class Warnings, trigger "PT_Avisos de servicio  1" bit 40
   66: '', class Warnings, trigger "PT_Avisos de servicio  1" bit 65
   2007: '', class Errors, trigger "PT_Acuses OP  1" bit 6
   2197: '', class Errors, trigger "PT_Acuses OP  2" bit 36
   2012: '', class Errors, trigger "PT_Acuses OP  1" bit 11
   2212: '', class Errors, trigger "PT_Acuses OP  2" bit 51
   42: '', class Warnings, trigger "PT_Avisos de servicio  1" bit 41
   2013: '', class Errors, trigger "PT_Acuses OP  1" bit 12
   2136: '', class Errors, trigger "PT_Acuses OP  1" bit 135
   2029: '', class Errors, trigger "PT_Acuses OP  1" bit 28
   26: '', class Warnings, trigger "PT_Avisos de servicio  1" bit 25
   2239: '', class Errors, trigger "PT_Acuses OP  2" bit 78
   2020: '', class Errors, trigger "PT_Acuses OP  1" bit 19
   2051: '', class Errors, trigger "PT_Acuses OP  1" bit 50
   2240: '', class Errors, trigger "PT_Acuses OP  2" bit 79
   28: '', class Warnings, trigger "PT_Avisos de servicio  1" bit 27
   2100: '', class Errors, trigger "PT_Acuses OP  1" bit 99
   2066: '', class Errors, trigger "PT_Acuses OP  1" bit 65
   2214: '', class Errors, trigger "PT_Acuses OP  2" bit 53
   64: '', class Warnings, trigger "PT_Avisos de servicio  1" bit 63
   2232: '', class Errors, trigger "PT_Acuses OP  2" bit 71
   14: '', class Warnings, trigger "PT_Avisos de servicio  1" bit 13
   59: '', class Warnings, trigger "PT_Avisos de servicio  1" bit 58
   2182: '', class Errors, trigger "PT_Acuses OP  2" bit 21
   2132: '', class Errors, trigger "PT_Acuses OP  1" bit 131
   2054: '', class Errors, trigger "PT_Acuses OP  1" bit 53
   2028: '', class Errors, trigger "PT_Acuses OP  1" bit 27
   18: '', class Warnings, trigger "PT_Avisos de servicio  1" bit 17
   2147: '', class Errors, trigger "PT_Acuses OP  1" bit 146
   2060: '', class Errors, trigger "PT_Acuses OP  1" bit 59
   2179: '', class Errors, trigger "PT_Acuses OP  2" bit 18
   2002: '', class Errors, trigger "PT_Acuses OP  1" bit 1
   47: '', class Warnings, trigger "PT_Avisos de servicio  1" bit 46
   23: '', class Warnings, trigger "PT_Avisos de servicio  1" bit 22
   2155: '', class Errors, trigger "PT_Acuses OP  1" bit 154
   2127: '', class Errors, trigger "PT_Acuses OP  1" bit 126
   2016: '', class Errors, trigger "PT_Acuses OP  1" bit 15
   2228: '', class Errors, trigger "PT_Acuses OP  2" bit 67
   2151: '', class Errors, trigger "PT_Acuses OP  1" bit 150
   2172: '', class Errors, trigger "PT_Acuses OP  2" bit 11
   2006: '', class Errors, trigger "PT_Acuses OP  1" bit 5
   54: '', class Warnings, trigger "PT_Avisos de servicio  1" bit 53
   2224: '', class Errors, trigger "PT_Acuses OP  2" bit 63
   2119: '', class Errors, trigger "PT_Acuses OP  1" bit 118
   36: '', class Warnings, trigger "PT_Avisos de servicio  1" bit 35
   2223: '', class Errors, trigger "PT_Acuses OP  2" bit 62

text list "ConvPsp": 0 ''; 1 ''

text list "Trasf_Tipe1": 0 ''; 1 ''

text list "Reset_kW": 0 ''; 1 ''

text list "Attendere2": 1 ''

text list "tipo_bobine": 0 ''; 1 ''; 2 ''; 3 ''; 4 ''; 5 ''

text list "CentoPercent": 0 ''; 1 ''; 2 ''; 3 ''; 4 ''; 5 ''; 6 ''; 7 ''; 8 ''; 9 ''; 10 ''; 11 ''

text list "Color8": 0 ''; 1 ''; 2 ''; 3 ''; 4 ''; 5 ''

text list "Imp_Exp": 0 ''; 1 ''

text list "BobTirVel": 0 ''; 1 ''

text list "Id_Sensor": 1 ''; 2 ''; 3 ''; 4 ''; 5 ''; 6 ''; 7 ''; 8 ''; 9 ''; 10 ''; 11 ''; 12 ''; 13 ''; 14 ''; 18 ''

text list "Color25": 0 ''; 1 ''; 2 ''; 3 ''; 4 ''; 5 ''

text list "ConvLun2": 0 ''; 1 ''

text list "T_Rosett": 0 ''

text list "SensInt1": 0 ''; 1 ''; 2 ''; 3 ''; 4 ''; 5 ''; 6 ''; 7 ''; 8 ''; 9 ''; 10 ''; 11 ''; 12 ''; 13 ''; 14 ''; 15 ''; 16 ''; 17 ''; 18 ''

text list "AGV": 0 ''; 1 ''; 2 ''; 3 ''; 4 ''; 5 ''; 6 ''; 7 ''; 8 ''; 9 ''; 10 ''; 11 ''; 12 ''; 13 ''; 14 ''; 15 ''; 16 ''; 17 ''; 18 ''

text list "Color4": 0 ''; 1 ''; 2 ''; 3 ''; 4 ''; 5 ''

text list "Color23": 0 ''; 1 ''; 2 ''; 3 ''; 4 ''; 5 ''

text list "Color19": 0 ''; 1 ''; 2 ''; 3 ''; 4 ''; 5 ''

text list "ConvKg": 0 ''; 1 ''

text list "Off_On2": 0 ''; 1 ''

text list "Sensor1": 2 ''; 3 ''; 4 ''; 5 ''; 6 ''; 7 ''; 8 ''

text list "Reset": 0 ''; 1 ''

text list "ConvEnergy": 0 ''; 1 ''

text list "ConvLun3": 0 ''; 1 ''

text list "SensInt2": 0 ''; 1 ''; 2 ''; 3 ''; 4 ''; 5 ''; 6 ''; 7 ''; 8 ''; 9 ''; 10 ''; 11 ''; 12 ''; 13 ''; 14 ''; 15 ''; 16 ''; 17 ''; 18 ''

text list "Rosett": 1 ''; 2 ''; 4 ''

text list "Richiesta": 0 ''; 1 ''

text list "Percentuale": 0 ''; 1 ''

text list "S_Rosett": 0 ''; 1 ''

text list "SensProp2": 0 ''; 1 ''; 2 ''; 3 ''; 4 ''; 5 ''; 6 ''; 7 ''; 8 ''; 9 ''; 10 ''; 11 ''; 12 ''; 13 ''; 14 ''; 15 ''; 16 ''; 17 ''; 18 ''

text list "Totalizz": 0 ''; 1 ''; 2 ''; 3 ''; 4 ''

text list "ConvLun1": 0 ''; 1 ''

text list "SensProp1": 0 ''; 1 ''; 2 ''; 3 ''; 4 ''; 5 ''; 6 ''; 7 ''; 8 ''; 9 ''; 10 ''; 11 ''; 12 ''; 13 ''; 14 ''; 15 ''; 16 ''; 17 ''; 18 ''

text list "LaserChoic": 0 ''; 1 ''

text list "_percento": 0 ''; 1 ''

text list "Mux": 0 ''; 1 ''; 2 ''; 3 ''; 4 ''; 5 ''

text list "Domanda": 1 ''

text list "OutTraf": 1 ''; 2 ''; 4 ''

text list "ConvProdm": 0 ''; 1 ''

text list "Recipe_Wait": 0 ''; 1 ''

text list "MemRall": 0 ''; 1 ''

text list "Stato_Linea": 0 ''; 1 ''; 2 ''; 3 ''; 4 ''; 5 ''; 6 ''; 7 ''; 8 ''; 9 ''; 10 ''

text list "Fast_jog": 1 ''; 2 ''; 3 ''; 4 ''; 5 ''; 6 ''; 7 ''; 8 ''; 9 ''; 10 ''; 11 ''; 12 ''; 13 ''; 14 ''; 15 ''; 16 ''; 17 ''; 18 ''

text list "Color2": 0 ''; 1 ''; 2 ''; 3 ''; 4 ''; 5 ''

text list "Color7": 0 ''; 1 ''; 2 ''; 3 ''; 4 ''; 5 ''

text list "Color18": 0 ''; 1 ''; 2 ''; 3 ''; 4 ''; 5 ''

text list "Diametro": 0 ''; 1 ''

text list "No_Sì": 0 ''; 1 ''

text list "Blocks1": 1 ''; 2 ''; 3 ''; 4 ''; 5 ''; 6 ''; 7 ''; 8 ''; 9 ''; 10 ''; 11 ''; 17 ''; 18 ''

text list "Sens_Offset": 1 ''; 2 ''; 3 ''; 4 ''; 5 ''; 6 ''; 7 ''; 8 ''; 9 ''; 10 ''; 11 ''; 12 ''; 13 ''; 14 ''; 15 ''; 16 ''; 17 ''; 18 ''

text list "Blocks": 1 ''; 2 ''; 3 ''; 4 ''; 5 ''; 6 ''; 7 ''; 8 ''; 9 ''; 10 ''; 11 ''; 12 ''; 13 ''; 14 ''; 15 ''; 16 ''; 17 ''; 18 ''

text list "Sel_count": 0 ''; 1 ''

text list "Color3": 0 ''; 1 ''; 2 ''; 3 ''; 4 ''; 5 ''

text list "Attesa": 1 ''

text list "OtoMotorized": 0 ''; 1 ''

text list "TiroVelocità": 0 ''; 1 ''

text list "Color6": 0 ''; 1 ''; 2 ''; 3 ''; 4 ''; 5 ''

text list "Par_Type": 0 ''; 128 ''

text list "Color24": 0 ''; 1 ''; 2 ''; 3 ''; 4 ''; 5 ''

text list "ConvTime": 0 ''; 1 ''

text list "ConvVel": 0 ''; 1 ''

text list "Elevat": 1 ''; 2 ''; 4 ''

text list "ConvTotm": 0 ''; 1 ''

text list "Attendere4": 0 ''; 1 ''; 2 ''

text list "Contametri": 0 ''; 1 ''; 2 ''

text list "Task_Id": 1 ''; 6 ''; 11 ''; 12 ''; 13 ''; 14 ''

text list "ConvSetm": 0 ''; 1 ''

text list "Color5": 0 ''; 1 ''; 2 ''; 3 ''; 4 ''; 5 ''

text list "ConvLun": 0 ''; 1 ''

text list "Color22": 0 ''; 1 ''; 2 ''; 3 ''; 4 ''; 5 ''

text list "SensIntTime": 0 ''; 1 ''; 2 ''; 3 ''; 4 ''; 5 ''; 6 ''; 7 ''; 8 ''; 9 ''; 10 ''; 11 ''; 12 ''; 13 ''; 14 ''; 15 ''; 16 ''; 17 ''; 18 ''

text list "Norm_OTO": 0 ''; 1 ''

text list "SensInt4": 0 ''; 1 ''; 2 ''; 3 ''; 4 ''; 5 ''; 6 ''; 7 ''; 8 ''; 9 ''; 10 ''; 11 ''; 12 ''; 13 ''; 14 ''; 15 ''; 16 ''; 17 ''; 18 ''

text list "Trasf_Tipe": 0 ''; 1 ''

text list "OutChoice": 1 ''; 2 ''; 4 ''

text list "Color20": 0 ''; 1 ''; 2 ''; 3 ''; 4 ''; 5 ''

text list "TiroVelocit1": 0 ''; 1 ''

text list "Oriz_Ver": 0 ''; 1 ''

text list "F6": 1 ''

text list "Die_Wear_Ch1": 0 ''; 1 ''; 2 ''; 3 ''

text list "Esc_Inc": 0 ''; 1 ''; 2 ''

text list "BobTV": 1 ''; 2 ''; 4 ''

text list "L_Pilota": 1 ''; 2 ''; 4 ''

text list "RoseStat": 0 ''; 1 ''; 2 ''

text list "Color1": 0 ''; 1 ''; 2 ''; 3 ''; 4 ''; 5 ''

text list "F4": 1 ''

text list "Sfilaggio": 0 ''; 1 ''

text list "Tiro": 0 ''; 1 ''

text list "Color17": 0 ''; 1 ''; 2 ''; 3 ''; 4 ''; 5 ''

text list "Attendere1": 1 ''

text list "Off_On": 0 ''; 1 ''

text list "L_Bob": 1 ''; 2 ''

text list "SBPM": 0 ''; 1 ''

text list "LaserAlCh": 0 ''; 1 ''

text list "LaserStato": 0 ''; 3 ''; 4 ''; 5 ''; 6 ''; 10 ''

text list "Attendere3": 1 ''

text list "Off_On3": 0 ''; 1 ''

text list "Bobina": 0 ''; 1 ''

text list "Color21": 0 ''; 1 ''; 2 ''; 3 ''; 4 ''; 5 ''

text list "Coppia": 0 ''; 1 ''

screen "Manteinance" 800x448, template "Template"
   GraphicView "Graphic_0" at 614,372 size 106x76
   TextField "OBJECT_2" at 92,369 size 248x32
   TextField "OBJECT_3" at 92,336 size 248x32
   TextField "OBJECT_4" at 92,68 size 264x32
   TextField "OBJECT_5" at 92,200 size 264x32
   TextField "OBJECT_6" at 92,167 size 264x32
   TextField "OBJECT_7" at 92,134 size 264x32
   TextField "OBJECT_8" at 92,101 size 264x32
   TextField "OBJECT_9" at 428,0 size 104x32
   TextField "OBJECT_10" at 476,35 size 88x32
   TextField "OBJECT_11" at 348,35 size 120x32
   IOField "OBJECT_12" at 348,369 size 152x16
   IOField "OBJECT_13" at 348,336 size 152x16
   IOField "OBJECT_14" at 364,68 size 104x16
   IOField "OBJECT_15" at 476,68 size 104x16
   IOField "OBJECT_16" at 364,101 size 104x16
   IOField "OBJECT_17" at 476,101 size 104x16
   SymbolicIOField "OBJECT_18" at 588,68 size 120x32
   IOField "OBJECT_19" at 364,134 size 104x16
   IOField "OBJECT_20" at 476,134 size 104x16
   SymbolicIOField "OBJECT_21" at 588,134 size 120x32
   SymbolicIOField "OBJECT_22" at 588,101 size 120x32
   IOField "OBJECT_23" at 364,167 size 104x16
   IOField "OBJECT_24" at 476,167 size 104x16
   SymbolicIOField "OBJECT_25" at 588,167 size 120x32
   IOField "OBJECT_26" at 364,200 size 104x16
   IOField "OBJECT_27" at 476,200 size 104x16
   SymbolicIOField "OBJECT_28" at 588,200 size 120x32

screen "Trend24" 800x448, template "Template"
   TextField "OBJECT_1" at 305,390 size 431x31
   TrendView "OBJECT_3" at 80,0 size 640x368
   IOField "Campo ES_1" at 185,392 size 118x32

screen "SetUpTech2" 800x448, template "Template"
   TextField "OBJECT_1" at 268,16 size 264x32
   TextField "OBJECT_3" at 92,80 size 264x32
   TextField "OBJECT_4" at 92,128 size 264x32
   TextField "OBJECT_5" at 92,176 size 264x32
   TextField "OBJECT_6" at 364,128 size 88x32
   TextField "OBJECT_7" at 540,128 size 88x32
   TextField "OBJECT_8" at 364,176 size 88x32
   TextField "OBJECT_9" at 540,176 size 88x32
   TextField "OBJECT_11" at 92,224 size 440x32
   TextField "OBJECT_34" at 92,272 size 440x32
   TextField "OBJECT_36" at 588,272 size 24x32
   IOField "OBJECT_13" at 364,80 size 88x32
   IOField "OBJECT_14" at 444,128 size 88x32
   IOField "OBJECT_15" at 620,128 size 88x32
   IOField "OBJECT_16" at 444,176 size 88x32
   IOField "OBJECT_17" at 620,176 size 88x32
   SymbolicIOField "OBJECT_18" at 524,224 size 184x44
   IOField "OBJECT_35" at 524,272 size 56x32

screen "Matassatore" 800x448, template "Template"
   TextField "OBJECT_6" at 332,32 size 184x32
   TextField "OBJECT_8" at 80,208 size 472x32
   TextField "OBJECT_30" at 652,208 size 56x32
   SymbolicIOField "OBJECT_22" at 80,144 size 472x32
   SymbolicIOField "OBJECT_23" at 652,144 size 24x32
   SymbolicIOField "OBJECT_24" at 80,96 size 472x32
   IOField "OBJECT_25" at 556,144 size 88x32
   SymbolicIOField "OBJECT_28" at 552,96 size 168x32
   IOField "OBJECT_14" at 556,208 size 88x32

screen "FreeParamet" 800x448, template "Template"
   TextField "OBJECT_1" at 124,384 size 456x32
   TextField "OBJECT_2" at 80,112 size 120x32
   TextField "OBJECT_3" at 80,64 size 280x32
   TextField "OBJECT_4" at 284,16 size 248x32
   TextField "OBJECT_5" at 80,160 size 296x32
   TextField "OBJECT_6" at 80,208 size 296x32
   TextField "OBJECT_7" at 476,208 size 216x32
   TextField "OBJECT_8" at 80,256 size 296x32
   TextField "OBJECT_9" at 80,304 size 136x32
   TextField "OBJECT_10" at 268,304 size 56x32
   TextField "OBJECT_11" at 492,304 size 56x32
   TextField "OBJECT_12" at 556,64 size 56x32
   SymbolicIOField "OBJECT_13" at 216,112 size 504x44
   SymbolicIOField "OBJECT_14" at 364,64 size 184x44
   IOField "OBJECT_15" at 620,64 size 40x32
   SymbolicIOField "OBJECT_16" at 396,160 size 24x44
   IOField "OBJECT_17" at 380,208 size 72x32
   IOField "OBJECT_18" at 380,256 size 72x32
   IOField "OBJECT_19" at 348,304 size 120x32
   IOField "OBJECT_20" at 572,304 size 120x32

screen "SetUpTech5" 800x448, template "Template"
   TextField "OBJECT_1" at 124,16 size 568x32
   TextField "OBJECT_34" at 80,96 size 312x32
   TextField "OBJECT_35" at 80,128 size 312x32
   TextField "OBJECT_36" at 80,160 size 312x32
   TextField "OBJECT_37" at 80,192 size 312x32
   TextField "OBJECT_38" at 80,224 size 312x32
   TextField "OBJECT_39" at 80,256 size 312x32
   TextField "OBJECT_40" at 396,256 size 42x31
   TextField "OBJECT_41" at 445,256 size 24x32
   TextField "OBJECT_42" at 445,224 size 24x32
   TextField "OBJECT_43" at 445,192 size 24x32
   TextField "OBJECT_44" at 445,160 size 24x32
   TextField "OBJECT_45" at 445,128 size 24x32
   TextField "OBJECT_51" at 80,304 size 472x32
   TextField "OBJECT_52" at 80,336 size 472x32
   TextField "OBJECT_55" at 604,304 size 40x32
   TextField "OBJECT_56" at 445,96 size 216x32
   IOField "OBJECT_46" at 396,96 size 34x33
   IOField "OBJECT_47" at 396,128 size 50x33
   IOField "OBJECT_48" at 396,160 size 50x33
   IOField "OBJECT_49" at 396,192 size 50x33
   IOField "OBJECT_50" at 396,224 size 50x33
   SymbolicIOField "OBJECT_53" at 540,336 size 56x44
   IOField "OBJECT_54" at 540,304 size 72x32

screen "Start" 800x448, template "Template"
   TextField "OBJECT_1" at 80,0 size 248x32
   TextField "OBJECT_2" at 80,32 size 200x32
   TextField "OBJECT_3" at 80,64 size 200x32
   TextField "OBJECT_4" at 80,96 size 200x32
   TextField "OBJECT_5" at 325,413 size 88x32
   TextField "OBJECT_6" at 528,387 size 104x48
   TextField "OBJECT_7" at 396,32 size 184x32
   TextField "OBJECT_8" at 80,416 size 104x32
   TextField "OBJECT_9" at 672,387 size 48x48
   TextField "OBJECT_73" at 371,64 size 56x32
   TextField "OBJECT_74" at 371,96 size 56x32
   TextField "OBJECT_75" at 339,32 size 56x32
   Bar "OBJECT_10" at 432,96 size 288x32
   Bar "OBJECT_11" at 432,64 size 288x32
   SymbolicIOField "OBJECT_12" at 456,0 size 264x32
   IOField "OBJECT_13" at 268,32 size 72x32
   SymbolicIOField "OBJECT_14" at 128,176 size 40x44
   SymbolicIOField "OBJECT_15" at 176,176 size 40x44
   SymbolicIOField "OBJECT_16" at 224,176 size 40x44
   SymbolicIOField "OBJECT_17" at 272,176 size 40x44
   SymbolicIOField "OBJECT_18" at 528,176 size 40x44
   SymbolicIOField "OBJECT_19" at 112,224 size 456x16
   SymbolicIOField "OBJECT_20" at 520,355 size 200x32
   IOField "OBJECT_21" at 348,259 size 168x32
   IOField "OBJECT_22" at 348,291 size 168x32
   IOField "OBJECT_23" at 348,323 size 168x32
   IOField "OBJECT_24" at 348,355 size 168x32
   IOField "OBJECT_25" at 348,387 size 168x32
   IOField "OBJECT_26" at 524,259 size 152x32
   IOField "OBJECT_27" at 524,291 size 152x32
   IOField "OBJECT_28" at 524,323 size 152x32
   SymbolicIOField "OBJECT_29" at 320,176 size 40x44
   SymbolicIOField "OBJECT_30" at 368,176 size 40x44
   SymbolicIOField "OBJECT_31" at 416,176 size 40x44
   IOField "OBJECT_32" at 268,64 size 104x32
   IOField "OBJECT_33" at 268,96 size 104x32
   IOField "OBJECT_34" at 183,428 size 142x17
   IOField "OBJECT_35" at 413,428 size 114x17
   IOField "OBJECT_36" at 624,387 size 48x48
   IOField "OBJECT_37" at 112,240 size 56x16
   IOField "OBJECT_38" at 160,240 size 56x16
   IOField "OBJECT_39" at 208,240 size 56x16
   IOField "OBJECT_40" at 256,240 size 56x16
   IOField "OBJECT_41" at 304,240 size 56x16
   IOField "OBJECT_42" at 352,240 size 56x16
   IOField "OBJECT_43" at 400,240 size 56x16
   SymbolicIOField "OBJECT_44" at 528,144 size 48x32
   IOField "OBJECT_45" at 512,240 size 56x16
   SymbolicIOField "OBJECT_49" at 128,144 size 40x32
   SymbolicIOField "OBJECT_50" at 176,144 size 40x32
   SymbolicIOField "OBJECT_51" at 224,144 size 40x32
   SymbolicIOField "OBJECT_52" at 272,144 size 40x32
   SymbolicIOField "OBJECT_53" at 320,144 size 40x32
   SymbolicIOField "OBJECT_54" at 368,144 size 40x32
   SymbolicIOField "OBJECT_55" at 416,144 size 40x32
   IOField "OBJECT_56" at 572,32 size 104x32
   SymbolicIOField "OBJECT_57" at 464,144 size 40x32
   SymbolicIOField "OBJECT_59" at 464,176 size 40x44
   IOField "OBJECT_61" at 448,240 size 56x16
   SymbolicIOField "OBJECT_63" at 316,0 size 120x32
   SymbolicIOField "OBJECT_64" at 664,32 size 56x32
   SymbolicIOField "OBJECT_65" at 80,259 size 280x32
   SymbolicIOField "OBJECT_66" at 80,291 size 280x32
   SymbolicIOField "OBJECT_67" at 80,323 size 280x32
   SymbolicIOField "OBJECT_68" at 80,355 size 280x32
   SymbolicIOField "OBJECT_69" at 80,387 size 280x32
   SymbolicIOField "OBJECT_70" at 677,259 size 40x32
   SymbolicIOField "OBJECT_71" at 677,291 size 40x32
   SymbolicIOField "OBJECT_72" at 677,323 size 40x32

screen "SetUpTech1" 800x448, template "Template"
   TextField "OBJECT_1" at 268,0 size 264x32
   TextField "OBJECT_2" at 80,32 size 280x32
   TextField "OBJECT_3" at 80,96 size 280x32
   TextField "OBJECT_4" at 80,160 size 280x32
   TextField "OBJECT_5" at 80,288 size 408x32
   TextField "OBJECT_6" at 80,352 size 296x32
   TextField "OBJECT_7" at 444,352 size 40x32
   TextField "OBJECT_8" at 80,384 size 216x32
   TextField "OBJECT_9" at 364,384 size 72x32
   TextField "OBJECT_10" at 80,416 size 360x32
   TextField "OBJECT_11" at 540,32 size 56x32
   TextField "OBJECT_12" at 80,64 size 280x32
   TextField "OBJECT_31" at 80,256 size 536x32
   TextField "OBJECT_33" at 684,256 size 24x32
   TextField "OBJECT_34" at 80,320 size 408x32
   TextField "OBJECT_38" at 80,128 size 280x32
   SymbolicIOField "OBJECT_13" at 348,32 size 184x36
   SymbolicIOField "OBJECT_14" at 348,96 size 120x36
   SymbolicIOField "OBJECT_15" at 348,160 size 184x32
   SymbolicIOField "OBJECT_16" at 344,192 size 376x32
   IOField "OBJECT_17" at 476,288 size 168x32
   IOField "OBJECT_18" at 364,352 size 88x32
   SymbolicIOField "OBJECT_19" at 284,384 size 56x32
   SymbolicIOField "OBJECT_20" at 428,384 size 56x32
   SymbolicIOField "OBJECT_21" at 363,415 size 56x32
   SymbolicIOField "OBJECT_22" at 460,96 size 216x32
   SymbolicIOField "OBJECT_23" at 345,224 size 40x32
   SymbolicIOField "OBJECT_24" at 529,160 size 136x32
   SymbolicIOField "OBJECT_25" at 664,159 size 56x32
   IOField "OBJECT_26" at 604,32 size 40x32
   SymbolicIOField "OBJECT_27" at 664,96 size 56x36
   IOField "OBJECT_28" at 348,67 size 40x32
   SymbolicIOField "OBJECT_29" at 80,192 size 265x32
   SymbolicIOField "OBJECT_30" at 80,224 size 265x32
   IOField "OBJECT_32" at 620,256 size 56x32
   IOField "OBJECT_35" at 476,320 size 168x32
   SymbolicIOField "OBJECT_37" at 348,128 size 40x36
   SymbolicIOField "OBJECT_39" at 460,128 size 216x32
   SymbolicIOField "OBJECT_40" at 664,128 size 56x36

screen "Trend6" 800x448, template "Template"
   TextField "OBJECT_1" at 208,401 size 417x31
   TrendView "OBJECT_3" at 66,4 size 649x387

screen "SetUpOperat" 800x448, template "Template"
   TextField "OBJECT_1" at 236,32 size 328x32
   TextField "OBJECT_3" at 80,96 size 504x32
   TextField "OBJECT_4" at 80,208 size 504x32
   TextField "OBJECT_5" at 172,144 size 24x32
   TextField "OBJECT_6" at 172,256 size 24x32
   TextField "OBJECT_47" at 204,144 size 216x32
   TextField "OBJECT_48" at 204,256 size 216x32
   IOField "OBJECT_11" at 80,144 size 88x32
   IOField "OBJECT_12" at 80,256 size 88x32

screen "SetUpTech6" 800x448, template "Template"
   TextField "OBJECT_1" at 80,16 size 640x32
   TextField "OBJECT_2" at 80,64 size 59x17
   TextField "OBJECT_3" at 80,80 size 59x17
   TextField "OBJECT_4" at 80,96 size 59x17
   TextField "OBJECT_19" at 316,64 size 24x32
   TextField "OBJECT_35" at 316,80 size 24x32
   TextField "OBJECT_36" at 316,96 size 24x32
   TextField "OBJECT_37" at 316,112 size 24x32
   TextField "OBJECT_38" at 316,128 size 24x32
   TextField "OBJECT_39" at 316,144 size 24x32
   TextField "OBJECT_40" at 316,160 size 24x32
   TextField "OBJECT_41" at 316,176 size 24x32
   TextField "OBJECT_42" at 316,192 size 24x32
   TextField "OBJECT_43" at 316,208 size 24x32
   TextField "OBJECT_44" at 316,224 size 24x32
   TextField "OBJECT_45" at 316,240 size 24x32
   TextField "OBJECT_46" at 316,256 size 24x32
   TextField "OBJECT_47" at 316,272 size 24x32
   TextField "OBJECT_48" at 316,288 size 24x32
   TextField "OBJECT_49" at 316,304 size 24x32
   TextField "OBJECT_50" at 80,128 size 59x17
   TextField "OBJECT_51" at 80,144 size 59x17
   TextField "OBJECT_52" at 80,112 size 59x17
   TextField "OBJECT_53" at 80,176 size 59x17
   TextField "OBJECT_54" at 80,192 size 59x17
   TextField "OBJECT_55" at 80,160 size 59x17
   TextField "OBJECT_56" at 80,224 size 63x17
   TextField "OBJECT_57" at 80,240 size 63x17
   TextField "OBJECT_58" at 80,208 size 63x17
   TextField "OBJECT_59" at 80,272 size 63x17
   TextField "OBJECT_60" at 80,288 size 63x17
   TextField "OBJECT_61" at 80,256 size 63x17
   TextField "OBJECT_62" at 80,304 size 63x17
   TextField "OBJECT_63" at 364,112 size 62x17
   TextField "OBJECT_64" at 524,64 size 88x32
   TextField "OBJECT_65" at 620,64 size 88x32
   TextField "OBJECT_66" at 364,128 size 62x17
   TextField "OBJECT_67" at 364,160 size 62x17
   TextField "OBJECT_68" at 364,144 size 62x17
   TextField "OBJECT_69" at 364,176 size 62x17
   TextField "OBJECT_70" at 364,192 size 62x17
   TextField "OBJECT_83" at 680,112 size 24x17
   TextField "OBJECT_84" at 680,128 size 24x17
   TextField "OBJECT_85" at 680,144 size 24x17
   TextField "OBJECT_86" at 680,160 size 24x17
   TextField "OBJECT_87" at 680,192 size 24x17
   TextField "OBJECT_88" at 680,176 size 24x17
   IOField "OBJECT_18" at 236,64 size 88x16
   IOField "OBJECT_20" at 236,80 size 88x16
   IOField "OBJECT_21" at 236,96 size 88x16
   IOField "OBJECT_22" at 236,112 size 88x16
   IOField "OBJECT_23" at 236,128 size 88x16
   IOField "OBJECT_24" at 236,144 size 88x16
   IOField "OBJECT_25" at 236,160 size 88x16
   IOField "OBJECT_26" at 236,176 size 88x16
   IOField "OBJECT_27" at 236,192 size 88x16
   IOField "OBJECT_28" at 236,208 size 88x16
   IOField "OBJECT_29" at 236,224 size 88x16
   IOField "OBJECT_30" at 236,240 size 88x16
   IOField "OBJECT_31" at 236,256 size 88x16
   IOField "OBJECT_32" at 236,272 size 88x16
   IOField "OBJECT_33" at 236,288 size 88x16
   IOField "OBJECT_34" at 236,304 size 88x16
   IOField "OBJECT_71" at 524,112 size 88x16
   IOField "OBJECT_72" at 604,112 size 88x16
   IOField "OBJECT_73" at 604,128 size 88x16
   IOField "OBJECT_74" at 524,128 size 88x16
   IOField "OBJECT_75" at 604,144 size 88x16
   IOField "OBJECT_76" at 524,144 size 88x16
   IOField "OBJECT_77" at 604,160 size 88x16
   IOField "OBJECT_78" at 524,160 size 88x16
   IOField "OBJECT_79" at 604,176 size 88x16
   IOField "OBJECT_80" at 524,176 size 88x16
   IOField "OBJECT_81" at 604,192 size 88x16
   IOField "OBJECT_82" at 524,192 size 88x16

screen "OTO" 800x448, template "Template"
   TextField "OBJECT_1" at 140,16 size 475x39
   TextField "OBJECT_2" at 104,80 size 100x54
   TextField "OBJECT_3" at 96,192 size 128x54
   TextField "OBJECT_4" at 96,304 size 94x54
   TextField "OBJECT_5" at 544,176 size 80x54
   TextField "OBJECT_11" at 540,96 size 99x27
   TextField "OBJECT_13" at 620,128 size 24x32
   Bar "OBJECT_6" at 288,80 size 208x320
   IOField "OBJECT_7" at 163,144 size 126x32
   IOField "OBJECT_8" at 162,256 size 126x32
   IOField "OBJECT_9" at 156,368 size 126x32
   IOField "OBJECT_10" at 572,256 size 72x32
   IOField "OBJECT_12" at 544,128 size 34x33

screen "Stratificato" 800x448, template "Template"
   TextField "OBJECT_2" at 284,16 size 232x32
   TextField "OBJECT_26" at 80,64 size 424x32
   TextField "OBJECT_28" at 604,64 size 72x32
   TextField "OBJECT_29" at 80,112 size 424x32
   TextField "OBJECT_30" at 80,160 size 424x32
   TextField "OBJECT_35" at 80,208 size 424x32
   TextField "OBJECT_37" at 588,112 size 72x32
   TextField "OBJECT_38" at 588,160 size 72x32
   IOField "OBJECT_27" at 508,64 size 88x32
   IOField "OBJECT_32" at 508,112 size 72x32
   IOField "OBJECT_34" at 508,160 size 72x32
   SymbolicIOField "OBJECT_36" at 508,208 size 104x44

screen "Svolgitore" 800x448, template "Template"
   TextField "OBJECT_6" at 348,16 size 120x32
   TextField "OBJECT_29" at 80,64 size 552x17
   TextField "OBJECT_30" at 80,96 size 552x17
   TextField "OBJECT_54" at 80,80 size 552x17
   TextField "OBJECT_45" at 688,80 size 40x17
   TextField "OBJECT_56" at 688,64 size 40x17
   TextField "OBJECT_58" at 92,256 size 184x32
   TextField "OBJECT_59" at 492,256 size 216x32
   TextField "OBJECT_61" at 645,304 size 40x17
   TextField "OBJECT_62" at 229,304 size 40x17
   TextField "OBJECT_89" at 80,112 size 376x17
   Bar "OBJECT_25" at 272,184 size 176x224
   IOField "OBJECT_26" at 364,416 size 72x16
   SymbolicIOField "OBJECT_27" at 332,144 size 152x16
   SymbolicIOField "OBJECT_28" at 332,160 size 136x16
   SymbolicIOField "OBJECT_53" at 632,96 size 97x17
   IOField "OBJECT_47" at 616,80 size 72x16
   IOField "OBJECT_55" at 632,64 size 56x16
   IOField "OBJECT_57" at 124,304 size 104x16
   IOField "OBJECT_60" at 540,304 size 104x16
   SymbolicIOField "OBJECT_90" at 456,112 size 273x17

screen "AdjustSensor" 800x448, template "Template"
   GraphicView "Graphic_0" at 320,128 size 176x96
   GraphicView "Graphic_1" at 160,80 size 90x52
   GraphicView "Graphic_2" at 160,160 size 90x48
   TextField "OBJECT_1" at 92,16 size 344x32
   TextField "OBJECT_64" at 92,272 size 216x32
   TextField "OBJECT_65" at 92,320 size 216x32
   SymbolicIOField "OBJECT_5" at 444,16 size 136x44
   SymbolicIOField "OBJECT_18" at 96,128 size 180x32
   IOField "OBJECT_15" at 416,80 size 116x32
   SymbolicIOField "OBJECT_27" at 92,400 size 424x32
   IOField "OBJECT_62" at 316,272 size 200x32
   IOField "OBJECT_63" at 316,320 size 200x32

screen "SetUpPID" 800x448, template "Template"
   TextField "OBJECT_1" at 92,48 size 312x32
   TextField "OBJECT_2" at 92,80 size 312x32
   TextField "OBJECT_3" at 300,400 size 168x32
   TextField "OBJECT_4" at 604,48 size 56x32
   SymbolicIOField "OBJECT_5" at 412,48 size 184x44
   SymbolicIOField "OBJECT_6" at 412,80 size 264x44
   IOField "OBJECT_7" at 668,48 size 40x32
   SymbolicIOField "OBJECT_16" at 412,128 size 216x32
   IOField "OBJECT_17" at 616,128 size 104x32
   SymbolicIOField "OBJECT_18" at 412,176 size 216x32
   SymbolicIOField "OBJECT_19" at 412,224 size 216x32
   IOField "OBJECT_20" at 616,176 size 104x32
   IOField "OBJECT_21" at 616,224 size 104x32
   SymbolicIOField "OBJECT_22" at 80,176 size 216x32
   IOField "OBJECT_24" at 300,176 size 120x32
   SymbolicIOField "OBJECT_26" at 395,1 size 328x32
   SymbolicIOField "OBJECT_27" at 80,1 size 297x32
   SymbolicIOField "OBJECT_28" at 508,368 size 88x32
   SymbolicIOField "OBJECT_29" at 508,402 size 88x32
   SymbolicIOField "OBJECT_30" at 300,368 size 200x27
   SymbolicIOField "OBJECT_31" at 80,224 size 216x32
   SymbolicIOField "OBJECT_32" at 80,272 size 216x32
   SymbolicIOField "OBJECT_33" at 80,128 size 216x32
   IOField "OBJECT_34" at 300,224 size 120x32
   IOField "OBJECT_35" at 300,272 size 104x32
   IOField "OBJECT_36" at 300,128 size 88x32

screen "Bobinatore1" 800x448, template "Template"
   TextField "OBJECT_36" at 156,64 size 504x32
   TextField "OBJECT_34" at 252,224 size 136x32
   TextField "OBJECT_37" at 124,128 size 568x32
   TextField "OBJECT_40" at 124,160 size 568x32
   SymbolicIOField "OBJECT_33" at 412,224 size 136x50
   SymbolicIOField "OBJECT_20" at 220,16 size 360x32

screen "Laser" 800x448, template "Template"
   TextField "OBJECT_12" at 80,0 size 280x32
   TextField "OBJECT_13" at 80,32 size 280x32
   TextField "OBJECT_17" at 80,272 size 280x32
   TextField "OBJECT_18" at 80,416 size 280x32
   TextField "OBJECT_27" at 492,32 size 40x32
   TextField "OBJECT_28" at 492,80 size 40x32
   TextField "OBJECT_30" at 492,272 size 40x32
   TextField "OBJECT_32" at 492,320 size 40x32
   TextField "OBJECT_34" at 492,368 size 40x32
   TextField "OBJECT_36" at 492,176 size 40x32
   TextField "OBJECT_38" at 80,128 size 280x32
   TextField "OBJECT_39" at 492,128 size 40x32
   TextField "OBJECT_41" at 80,80 size 280x32
   TextField "OBJECT_42" at 80,176 size 280x32
   TextField "OBJECT_43" at 80,224 size 280x32
   TextField "OBJECT_44" at 80,320 size 280x32
   TextField "OBJECT_45" at 80,368 size 280x32
   SymbolicIOField "OBJECT_23" at 364,0 size 344x16
   SymbolicIOField "OBJECT_24" at 364,224 size 168x44
   SymbolicIOField "OBJECT_25" at 364,400 size 216x44
   IOField "OBJECT_26" at 364,32 size 120x32
   IOField "OBJECT_29" at 364,80 size 120x32
   IOField "OBJECT_31" at 364,272 size 120x32
   IOField "OBJECT_33" at 364,368 size 120x32
   IOField "OBJECT_35" at 364,320 size 120x32
   IOField "OBJECT_37" at 364,176 size 120x32
   IOField "OBJECT_40" at 364,128 size 120x32

screen "SetUpTech4" 800x448, template "Template"
   TextField "OBJECT_1" at 188,80 size 120x32
   TextField "OBJECT_2" at 108,16 size 584x32
   TextField "OBJECT_3" at 92,176 size 24x32
   TextField "OBJECT_4" at 92,144 size 24x32
   TextField "OBJECT_5" at 92,208 size 24x32
   TextField "OBJECT_6" at 92,240 size 24x32
   TextField "OBJECT_7" at 92,272 size 24x32
   TextField "OBJECT_8" at 92,304 size 24x32
   TextField "OBJECT_9" at 604,80 size 104x32
   TextField "OBJECT_10" at 316,80 size 104x32
   TextField "OBJECT_11" at 428,80 size 152x32
   TextField "OBJECT_13" at 92,80 size 88x32
   TextField "OBJECT_14" at 684,160 size 24x32
   TextField "OBJECT_15" at 684,192 size 24x32
   TextField "OBJECT_16" at 684,224 size 24x32
   TextField "OBJECT_17" at 684,256 size 24x32
   TextField "OBJECT_18" at 684,288 size 24x32
   TextField "OBJECT_19" at 684,320 size 24x32
   TextField "OBJECT_52" at 92,368 size 24x32
   TextField "OBJECT_53" at 92,336 size 24x32
   TextField "OBJECT_54" at 92,400 size 24x32
   TextField "OBJECT_55" at 684,352 size 24x32
   TextField "OBJECT_56" at 684,384 size 24x32
   IOField "OBJECT_20" at 188,144 size 88x32
   IOField "OBJECT_21" at 188,176 size 88x32
   IOField "OBJECT_22" at 188,208 size 88x32
   IOField "OBJECT_23" at 188,240 size 88x32
   IOField "OBJECT_24" at 188,272 size 88x32
   IOField "OBJECT_25" at 188,304 size 88x32
   IOField "OBJECT_26" at 604,160 size 72x32
   IOField "OBJECT_27" at 604,192 size 72x32
   IOField "OBJECT_28" at 604,224 size 72x32
   IOField "OBJECT_29" at 604,256 size 72x32
   IOField "OBJECT_30" at 604,288 size 72x32
   IOField "OBJECT_31" at 316,144 size 104x32
   IOField "OBJECT_32" at 316,176 size 104x32
   IOField "OBJECT_33" at 316,208 size 104x32
   IOField "OBJECT_34" at 316,240 size 104x32
   IOField "OBJECT_35" at 316,272 size 104x32
   IOField "OBJECT_36" at 428,144 size 104x32
   IOField "OBJECT_37" at 428,176 size 104x32
   IOField "OBJECT_38" at 428,208 size 104x32
   IOField "OBJECT_39" at 428,240 size 104x32
   IOField "OBJECT_40" at 428,272 size 104x32
   IOField "OBJECT_41" at 428,304 size 104x32
   IOField "OBJECT_42" at 316,304 size 104x32
   IOField "OBJECT_43" at 604,320 size 72x32
   SymbolicIOField "OBJECT_46" at 540,144 size 56x32
   SymbolicIOField "OBJECT_47" at 540,176 size 56x32
   SymbolicIOField "OBJECT_48" at 540,208 size 56x32
   SymbolicIOField "OBJECT_49" at 540,240 size 56x32
   SymbolicIOField "OBJECT_50" at 540,272 size 56x32
   SymbolicIOField "OBJECT_51" at 540,304 size 56x32
   IOField "OBJECT_57" at 188,336 size 88x32
   IOField "OBJECT_58" at 188,368 size 88x32
   IOField "OBJECT_59" at 188,400 size 88x32
   IOField "OBJECT_60" at 604,352 size 72x32
   IOField "OBJECT_61" at 604,384 size 72x32
   IOField "OBJECT_62" at 316,336 size 104x32
   IOField "OBJECT_63" at 316,368 size 104x32
   IOField "OBJECT_64" at 316,400 size 104x32
   IOField "OBJECT_65" at 428,336 size 104x32
   IOField "OBJECT_66" at 428,368 size 104x32
   IOField "OBJECT_67" at 428,400 size 104x32
   SymbolicIOField "OBJECT_68" at 540,336 size 56x32
   SymbolicIOField "OBJECT_69" at 540,368 size 56x32
   SymbolicIOField "OBJECT_70" at 540,400 size 56x32

screen "SetUpTech" 800x448, template "Template"
   TextField "OBJECT_1" at 284,16 size 232x32
   TextField "OBJECT_2" at 92,64 size 328x32
   TextField "OBJECT_3" at 92,144 size 392x32
   TextField "OBJECT_4" at 92,176 size 392x32
   TextField "OBJECT_5" at 92,208 size 392x32
   TextField "OBJECT_6" at 92,368 size 232x32
   TextField "OBJECT_7" at 92,400 size 232x32
   TextField "OBJECT_8" at 92,336 size 232x32
   TextField "OBJECT_9" at 488,288 size 232x32
   TextField "OBJECT_10" at 492,320 size 168x32
   TextField "OBJECT_12" at 412,336 size 24x32
   TextField "OBJECT_13" at 412,368 size 24x32
   TextField "OBJECT_14" at 412,400 size 24x32
   TextField "OBJECT_27" at 92,240 size 392x32
   IOField "OBJECT_15" at 332,336 size 72x32
   IOField "OBJECT_16" at 332,368 size 72x32
   IOField "OBJECT_17" at 332,400 size 72x32
   IOField "OBJECT_18" at 492,144 size 104x32
   IOField "OBJECT_19" at 492,176 size 104x32
   IOField "OBJECT_20" at 492,208 size 104x32
   SymbolicIOField "OBJECT_21" at 428,64 size 264x44
   SymbolicIOField "OBJECT_22" at 428,96 size 248x32
   SymbolicIOField "OBJECT_24" at 604,144 size 56x32
   SymbolicIOField "OBJECT_25" at 604,176 size 56x32
   SymbolicIOField "OBJECT_26" at 604,208 size 56x32
   IOField "OBJECT_28" at 492,240 size 104x32
   SymbolicIOField "OBJECT_29" at 604,240 size 56x32

screen "SetUpDrive" 800x448, template "Template"
   TextField "OBJECT_1" at 92,48 size 312x32
   TextField "OBJECT_2" at 92,80 size 312x32
   TextField "OBJECT_3" at 80,128 size 216x32
   TextField "OBJECT_5" at 412,176 size 216x32
   TextField "OBJECT_6" at 412,224 size 216x32
   TextField "OBJECT_7" at 412,272 size 216x32
   TextField "OBJECT_8" at 412,128 size 216x32
   TextField "OBJECT_9" at 80,400 size 168x32
   TextField "OBJECT_10" at 604,48 size 56x32
   TextField "OBJECT_28" at 80,272 size 216x32
   TextField "OBJECT_29" at 80,320 size 216x32
   SymbolicIOField "OBJECT_11" at 412,48 size 184x44
   SymbolicIOField "OBJECT_12" at 412,80 size 264x44
   IOField "OBJECT_13" at 668,48 size 40x32
   IOField "OBJECT_14" at 312,128 size 95x32
   IOField "OBJECT_15" at 312,176 size 95x32
   IOField "OBJECT_16" at 312,224 size 95x33
   IOField "OBJECT_17" at 616,176 size 104x32
   IOField "OBJECT_18" at 616,224 size 104x32
   IOField "OBJECT_19" at 616,272 size 72x32
   IOField "OBJECT_20" at 616,128 size 72x32
   SymbolicIOField "OBJECT_21" at 392,0 size 328x32
   SymbolicIOField "OBJECT_22" at 80,0 size 376x32
   SymbolicIOField "OBJECT_23" at 508,368 size 88x32
   SymbolicIOField "OBJECT_24" at 508,400 size 88x32
   SymbolicIOField "OBJECT_25" at 300,368 size 200x32
   SymbolicIOField "OBJECT_26" at 80,224 size 216x32
   SymbolicIOField "OBJECT_27" at 80,176 size 232x32
   IOField "OBJECT_30" at 312,271 size 95x32
   IOField "OBJECT_31" at 312,320 size 95x32

screen "Wear_Die" 800x448, template "Template"
   TextField "OBJECT_3" at 600,96 size 42x34
   TextField "OBJECT_5" at 511,59 size 24x16
   TextField "OBJECT_6" at 684,160 size 24x32
   TextField "OBJECT_7" at 684,192 size 24x32
   TextField "OBJECT_8" at 684,224 size 24x32
   TextField "OBJECT_9" at 684,256 size 24x32
   TextField "OBJECT_13" at 291,96 size 168x34
   TextField "OBJECT_72" at 511,75 size 24x16
   TextField "OBJECT_10" at 684,384 size 24x32
   TextField "OBJECT_73" at 684,288 size 24x32
   TextField "OBJECT_74" at 684,320 size 24x32
   TextField "OBJECT_87" at 684,352 size 24x32
   TextField "OBJECT_100" at 124,96 size 168x34
   TextField "OBJECT_101" at 444,96 size 152x34
   TextField "OBJECT_102" at 80,48 size 143x17
   TextField "OBJECT_104" at 80,16 size 149x17
   TextField "OBJECT_105" at 80,64 size 142x17
   IOField "OBJECT_15" at 439,75 size 72x16
   SymbolicIOField "OBJECT_16" at 440,16 size 280x44
   SymbolicIOField "OBJECT_17" at 80,144 size 40x32
   SymbolicIOField "OBJECT_18" at 80,176 size 40x32
   SymbolicIOField "OBJECT_19" at 80,208 size 40x32
   SymbolicIOField "OBJECT_20" at 80,240 size 40x32
   SymbolicIOField "OBJECT_21" at 80,272 size 40x32
   IOField "OBJECT_23" at 124,144 size 104x32
   IOField "OBJECT_24" at 284,144 size 104x32
   IOField "OBJECT_25" at 444,144 size 104x32
   IOField "OBJECT_26" at 124,176 size 104x32
   IOField "OBJECT_27" at 284,176 size 104x32
   IOField "OBJECT_28" at 444,176 size 104x32
   IOField "OBJECT_29" at 124,208 size 104x32
   IOField "OBJECT_30" at 284,208 size 104x32
   IOField "OBJECT_31" at 444,208 size 104x32
   IOField "OBJECT_32" at 124,240 size 104x32
   IOField "OBJECT_33" at 284,240 size 104x32
   IOField "OBJECT_34" at 444,240 size 104x32
   IOField "OBJECT_35" at 124,272 size 104x32
   IOField "OBJECT_36" at 284,272 size 104x32
   IOField "OBJECT_37" at 444,272 size 104x32
   IOField "OBJECT_42" at 604,160 size 72x32
   IOField "OBJECT_43" at 604,192 size 72x32
   IOField "OBJECT_44" at 604,256 size 72x32
   IOField "OBJECT_45" at 604,224 size 72x32
   SymbolicIOField "OBJECT_50" at 228,144 size 56x32
   SymbolicIOField "OBJECT_51" at 388,144 size 56x32
   SymbolicIOField "OBJECT_52" at 548,144 size 56x32
   SymbolicIOField "OBJECT_53" at 228,176 size 56x32
   SymbolicIOField "OBJECT_54" at 228,208 size 56x32
   SymbolicIOField "OBJECT_55" at 228,240 size 56x32
   SymbolicIOField "OBJECT_56" at 228,272 size 56x32
   SymbolicIOField "OBJECT_58" at 388,176 size 56x32
   SymbolicIOField "OBJECT_59" at 388,208 size 56x32
   SymbolicIOField "OBJECT_60" at 388,240 size 56x32
   SymbolicIOField "OBJECT_61" at 388,272 size 56x32
   SymbolicIOField "OBJECT_63" at 548,176 size 56x32
   SymbolicIOField "OBJECT_64" at 548,208 size 56x32
   SymbolicIOField "OBJECT_65" at 548,240 size 56x32
   SymbolicIOField "OBJECT_66" at 548,272 size 56x32
   IOField "OBJECT_71" at 439,59 size 72x16
   SymbolicIOField "OBJECT_88" at 80,368 size 40x32
   SymbolicIOField "OBJECT_22" at 80,400 size 40x32
   IOField "OBJECT_89" at 124,368 size 104x32
   IOField "OBJECT_90" at 284,368 size 104x32
   IOField "OBJECT_91" at 444,368 size 104x32
   IOField "OBJECT_40" at 444,400 size 104x32
   IOField "OBJECT_46" at 604,384 size 72x32
   SymbolicIOField "OBJECT_92" at 228,368 size 56x32
   SymbolicIOField "OBJECT_93" at 388,368 size 56x32
   SymbolicIOField "OBJECT_94" at 548,368 size 56x32
   SymbolicIOField "OBJECT_67" at 548,400 size 56x32
   SymbolicIOField "OBJECT_95" at 80,304 size 40x32
   IOField "OBJECT_96" at 124,304 size 104x32
   IOField "OBJECT_97" at 284,304 size 104x32
   IOField "OBJECT_98" at 444,304 size 104x32
   IOField "OBJECT_75" at 604,288 size 72x32
   IOField "OBJECT_76" at 604,320 size 72x32
   SymbolicIOField "OBJECT_77" at 228,304 size 56x32
   SymbolicIOField "OBJECT_78" at 388,304 size 56x32
   SymbolicIOField "OBJECT_79" at 548,304 size 56x32
   SymbolicIOField "OBJECT_80" at 548,336 size 56x32
   SymbolicIOField "OBJECT_81" at 80,336 size 40x32
   IOField "OBJECT_82" at 124,336 size 104x32
   SymbolicIOField "OBJECT_83" at 228,336 size 56x32
   IOField "OBJECT_84" at 284,336 size 104x32
   SymbolicIOField "OBJECT_85" at 388,336 size 56x32
   IOField "OBJECT_86" at 444,336 size 104x32
   IOField "OBJECT_99" at 604,352 size 72x32

screen "Logo" 800x448, template "Template"
   GraphicView "Graphic_0" at 290,50 size 224x222
   TextField "OBJECT_2" at 252,320 size 296x32
   TextField "OBJECT_3" at 236,368 size 328x32

screen "SetUpOperat2" 800x448, template "Template"
   TextField "OBJECT_27" at 252,32 size 312x32
   TextField "OBJECT_39" at 80,96 size 456x32
   TextField "OBJECT_40" at 80,128 size 456x32
   TextField "OBJECT_41" at 80,160 size 456x32
   TextField "OBJECT_42" at 80,192 size 456x32
   TextField "OBJECT_43" at 80,224 size 456x32
   TextField "OBJECT_44" at 80,256 size 456x32
   TextField "OBJECT_45" at 80,288 size 456x32
   TextField "OBJECT_46" at 80,320 size 456x32
   SymbolicIOField "OBJECT_16" at 540,192 size 38x35
   SymbolicIOField "OBJECT_17" at 540,160 size 38x35
   SymbolicIOField "OBJECT_18" at 540,128 size 38x35
   SymbolicIOField "OBJECT_19" at 540,224 size 38x35
   SymbolicIOField "OBJECT_20" at 540,256 size 38x35
   SymbolicIOField "OBJECT_21" at 540,288 size 38x35
   SymbolicIOField "OBJECT_22" at 540,320 size 38x35
   SymbolicIOField "OBJECT_38" at 540,96 size 38x35

screen "SetUpOperat3" 800x448, template "Template"
   TextField "OBJECT_2" at 80,64 size 472x32
   TextField "OBJECT_27" at 220,16 size 360x32
   TextField "OBJECT_29" at 80,96 size 472x32
   TextField "OBJECT_30" at 80,160 size 472x32
   TextField "OBJECT_31" at 80,128 size 472x32
   TextField "OBJECT_32" at 80,224 size 472x32
   TextField "OBJECT_33" at 80,288 size 472x32
   TextField "OBJECT_34" at 80,256 size 472x32
   TextField "OBJECT_35" at 80,192 size 472x32
   TextField "OBJECT_36" at 80,352 size 472x32
   TextField "OBJECT_37" at 80,416 size 472x32
   TextField "OBJECT_38" at 80,384 size 472x32
   TextField "OBJECT_39" at 80,320 size 472x32
   SymbolicIOField "OBJECT_15" at 556,64 size 38x35
   SymbolicIOField "OBJECT_16" at 556,160 size 38x35
   SymbolicIOField "OBJECT_17" at 556,128 size 38x35
   SymbolicIOField "OBJECT_18" at 556,96 size 38x35
   SymbolicIOField "OBJECT_19" at 556,192 size 38x35
   SymbolicIOField "OBJECT_20" at 556,224 size 38x35
   SymbolicIOField "OBJECT_21" at 556,256 size 38x35
   SymbolicIOField "OBJECT_22" at 556,288 size 38x35
   SymbolicIOField "OBJECT_23" at 556,320 size 38x35
   SymbolicIOField "OBJECT_25" at 556,384 size 38x35
   SymbolicIOField "OBJECT_26" at 556,352 size 38x35
   SymbolicIOField "OBJECT_28" at 556,417 size 38x35

screen "Dati2" 800x448, template "Template"
   TextField "OBJECT_3" at 108,64 size 24x32
   TextField "OBJECT_4" at 188,64 size 24x32
   TextField "OBJECT_5" at 252,64 size 40x32
   TextField "OBJECT_6" at 332,64 size 40x32
   TextField "OBJECT_27" at 412,64 size 40x32
   TextField "OBJECT_31" at 492,64 size 40x32
   Bar "OBJECT_7" at 576,128 size 32x276
   Bar "OBJECT_9" at 96,128 size 32x276
   Bar "OBJECT_10" at 176,128 size 32x276
   Bar "OBJECT_11" at 256,128 size 32x276
   Bar "OBJECT_12" at 336,128 size 32x276
   Bar "OBJECT_30" at 416,128 size 32x276
   Bar "OBJECT_34" at 496,128 size 32x276
   IOField "OBJECT_13" at 556,416 size 56x16
   SymbolicIOField "OBJECT_14" at 172,16 size 456x44
   SymbolicIOField "OBJECT_17" at 556,112 size 72x16
   SymbolicIOField "OBJECT_18" at 572,64 size 56x44
   SymbolicIOField "OBJECT_19" at 80,112 size 72x16
   SymbolicIOField "OBJECT_20" at 156,112 size 72x16
   IOField "OBJECT_21" at 80,416 size 56x16
   IOField "OBJECT_22" at 156,416 size 56x16
   SymbolicIOField "OBJECT_23" at 236,112 size 72x16
   IOField "OBJECT_24" at 236,416 size 56x16
   SymbolicIOField "OBJECT_25" at 316,112 size 72x16
   IOField "OBJECT_26" at 316,416 size 56x16
   SymbolicIOField "OBJECT_28" at 396,112 size 72x16
   IOField "OBJECT_29" at 396,416 size 56x16
   SymbolicIOField "OBJECT_32" at 476,112 size 72x16
   IOField "OBJECT_33" at 476,416 size 56x16

screen "Dati" 800x448, template "Template"
   TextField "OBJECT_1" at 140,64 size 24x32
   TextField "OBJECT_2" at 204,64 size 24x32
   TextField "OBJECT_3" at 268,64 size 24x32
   TextField "OBJECT_4" at 332,64 size 24x32
   TextField "OBJECT_5" at 396,64 size 24x32
   TextField "OBJECT_6" at 460,64 size 24x32
   TextField "OBJECT_7" at 524,64 size 24x32
   TextField "OBJECT_8" at 588,64 size 24x32
   Bar "OBJECT_10" at 192,128 size 30x278
   Bar "OBJECT_11" at 256,128 size 30x276
   Bar "OBJECT_12" at 320,128 size 32x276
   Bar "OBJECT_13" at 640,128 size 32x276
   Bar "OBJECT_14" at 126,128 size 30x278
   Bar "OBJECT_15" at 384,128 size 32x276
   Bar "OBJECT_16" at 448,128 size 32x276
   Bar "OBJECT_17" at 512,128 size 32x276
   Bar "OBJECT_18" at 576,128 size 32x276
   IOField "OBJECT_20" at 620,416 size 56x16
   SymbolicIOField "OBJECT_21" at 172,16 size 456x44
   IOField "OBJECT_22" at 108,416 size 56x16
   IOField "OBJECT_23" at 172,416 size 56x16
   IOField "OBJECT_24" at 236,416 size 56x16
   IOField "OBJECT_25" at 300,416 size 56x16
   IOField "OBJECT_26" at 364,416 size 56x16
   IOField "OBJECT_27" at 428,416 size 56x16
   IOField "OBJECT_28" at 492,416 size 56x16
   SymbolicIOField "OBJECT_29" at 108,112 size 72x16
   SymbolicIOField "OBJECT_30" at 172,112 size 72x16
   SymbolicIOField "OBJECT_31" at 236,112 size 72x16
   SymbolicIOField "OBJECT_32" at 300,112 size 72x16
   SymbolicIOField "OBJECT_33" at 492,112 size 72x16
   SymbolicIOField "OBJECT_34" at 428,112 size 72x16
   SymbolicIOField "OBJECT_35" at 620,112 size 72x16
   SymbolicIOField "OBJECT_36" at 364,112 size 72x16
   SymbolicIOField "OBJECT_37" at 636,64 size 56x44
   SymbolicIOField "OBJECT_38" at 556,112 size 72x16
   IOField "OBJECT_40" at 556,416 size 56x16

screen "Dati1" 800x448, template "Template"
   TextField "OBJECT_2" at 204,64 size 24x32
   TextField "OBJECT_3" at 268,64 size 24x32
   TextField "OBJECT_4" at 332,64 size 24x32
   TextField "OBJECT_5" at 396,64 size 24x32
   TextField "OBJECT_6" at 460,64 size 24x32
   TextField "OBJECT_7" at 524,64 size 24x32
   TextField "OBJECT_27" at 588,64 size 24x32
   Bar "OBJECT_8" at 256,128 size 30x278
   Bar "OBJECT_9" at 320,128 size 30x276
   Bar "OBJECT_10" at 384,128 size 32x276
   Bar "OBJECT_11" at 190,128 size 30x278
   Bar "OBJECT_12" at 448,128 size 32x276
   Bar "OBJECT_13" at 512,128 size 32x276
   Bar "OBJECT_28" at 576,128 size 32x276
   Bar "OBJECT_42" at 110,128 size 30x278
   SymbolicIOField "OBJECT_14" at 172,16 size 456x44
   IOField "OBJECT_15" at 172,416 size 56x16
   IOField "OBJECT_16" at 236,416 size 56x16
   IOField "OBJECT_17" at 300,416 size 56x16
   IOField "OBJECT_18" at 364,416 size 56x16
   IOField "OBJECT_19" at 428,416 size 56x16
   IOField "OBJECT_20" at 492,416 size 56x16
   SymbolicIOField "OBJECT_21" at 156,112 size 72x16
   SymbolicIOField "OBJECT_22" at 236,112 size 72x16
   SymbolicIOField "OBJECT_23" at 300,112 size 72x16
   SymbolicIOField "OBJECT_24" at 364,112 size 72x16
   SymbolicIOField "OBJECT_25" at 492,112 size 72x16
   SymbolicIOField "OBJECT_26" at 428,112 size 72x16
   IOField "OBJECT_29" at 556,416 size 56x16
   SymbolicIOField "OBJECT_30" at 556,112 size 72x16
   IOField "OBJECT_43" at 92,416 size 56x16
   SymbolicIOField "OBJECT_44" at 92,112 size 72x16
   SymbolicIOField "OBJECT_45" at 92,64 size 56x44

screen "SetUpTech3" 800x448, template "Template"
   TextField "OBJECT_1" at 268,16 size 264x32
   TextField "OBJECT_23" at 108,64 size 408x32
   TextField "OBJECT_34" at 108,112 size 408x32
   TextField "OBJECT_35" at 108,144 size 408x32
   TextField "OBJECT_36" at 108,208 size 408x32
   TextField "OBJECT_37" at 108,176 size 408x32
   TextField "OBJECT_38" at 108,272 size 408x32
   TextField "OBJECT_39" at 108,240 size 408x32
   IOField "OBJECT_14" at 524,112 size 104x32
   IOField "OBJECT_20" at 524,144 size 104x32
   IOField "OBJECT_21" at 524,176 size 104x32
   IOField "OBJECT_24" at 524,64 size 104x32
   IOField "OBJECT_26" at 524,208 size 104x32
   IOField "OBJECT_27" at 524,240 size 104x32
   IOField "OBJECT_29" at 524,272 size 104x32

screen "Trend12" 800x448, template "Template"
   TextField "OBJECT_1" at 211,395 size 442x32
   TrendView "OBJECT_3" at 80,0 size 640x368

screen "Bobinatore" 800x448, template "Template"
   Bar "OBJECT_8" at 208,60 size 512x80
   Bar "OBJECT_9" at 80,176 size 176x224
   Bar "OBJECT_10" at 448,176 size 176x224
   Bar "OBJECT_25" at 256,176 size 176x224
   IOField "OBJECT_12" at 96,64 size 88x32
   IOField "OBJECT_13" at 204,400 size 72x32
   IOField "OBJECT_14" at 544,400 size 72x32
   SymbolicIOField "OBJECT_18" at 80,64 size 72x32
   SymbolicIOField "OBJECT_19" at 96,16 size 80x42
   SymbolicIOField "OBJECT_20" at 220,16 size 506x31
   SymbolicIOField "OBJECT_21" at 492,144 size 168x16
   SymbolicIOField "OBJECT_22" at 492,160 size 152x16
   SymbolicIOField "OBJECT_23" at 96,96 size 114x31
   SymbolicIOField "OBJECT_24" at 96,128 size 91x31
   IOField "OBJECT_26" at 384,400 size 72x32
   SymbolicIOField "OBJECT_27" at 332,127 size 120x32
   SymbolicIOField "OBJECT_28" at 336,159 size 84x31

screen "Recipes" 800x448, template "Template"
   GraphicView "Graphic_0" at 614,372 size 106x76
   TextField "OBJECT_2" at 268,0 size 264x32
   TextField "OBJECT_3" at 92,48 size 264x32
   TextField "OBJECT_4" at 92,96 size 184x32
   IOField "OBJECT_5" at 364,48 size 40x32
   SymbolicIOField "OBJECT_6" at 284,96 size 168x44
   SymbolicIOField "OBJECT_7" at 492,96 size 40x44
   SymbolicIOField "OBJECT_8" at 556,96 size 152x32

screen "SetUpChief" 800x448, template "Template"
   TextField "OBJECT_1" at 236,16 size 328x32
   TextField "OBJECT_2" at 80,160 size 328x32
   TextField "OBJECT_5" at 80,80 size 312x32
   TextField "OBJECT_7" at 80,288 size 328x32
   TextField "OBJECT_8" at 80,320 size 328x32
   TextField "OBJECT_9" at 80,192 size 328x32
   TextField "OBJECT_10" at 80,224 size 328x32
   TextField "OBJECT_11" at 80,384 size 328x32
   TextField "OBJECT_12" at 80,352 size 328x32
   TextField "OBJECT_13" at 80,416 size 328x32
   TextField "OBJECT_34" at 80,256 size 328x32
   TextField "OBJECT_37" at 588,256 size 24x32
   TextField "OBJECT_40" at 396,112 size 72x32
   TextField "OBJECT_41" at 396,80 size 72x32
   IOField "OBJECT_15" at 460,80 size 72x32
   IOField "OBJECT_16" at 460,112 size 72x32
   SymbolicIOField "OBJECT_19" at 396,160 size 296x44
   SymbolicIOField "OBJECT_20" at 396,192 size 280x44
   IOField "OBJECT_22" at 396,320 size 72x32
   SymbolicIOField "OBJECT_23" at 396,224 size 168x44
   SymbolicIOField "OBJECT_24" at 396,352 size 56x44
   IOField "OBJECT_25" at 396,384 size 168x32
   IOField "OBJECT_26" at 396,416 size 136x32
   IOField "OBJECT_27" at 468,288 size 72x32
   SymbolicIOField "OBJECT_28" at 533,112 size 56x32
   SymbolicIOField "OBJECT_29" at 533,80 size 56x32
   SymbolicIOField "OBJECT_32" at 540,288 size 72x32
   SymbolicIOField "OBJECT_21" at 396,288 size 72x32
   SymbolicIOField "OBJECT_33" at 468,320 size 72x32
   IOField "OBJECT_35" at 397,256 size 104x32
   SymbolicIOField "OBJECT_36" at 502,256 size 104x32

screen "StratifTech" 800x448, template "Template"
   TextField "OBJECT_2" at 220,16 size 360x32
   TextField "OBJECT_11" at 80,64 size 424x32
   TextField "OBJECT_12" at 80,112 size 424x32
   TextField "OBJECT_15" at 80,160 size 424x32
   TextField "OBJECT_17" at 80,256 size 424x32
   TextField "OBJECT_19" at 588,64 size 40x32
   TextField "OBJECT_21" at 588,160 size 40x32
   TextField "OBJECT_22" at 588,112 size 40x32
   TextField "OBJECT_23" at 80,208 size 424x32
   TextField "OBJECT_24" at 588,208 size 40x32
   TextField "OBJECT_26" at 80,304 size 424x32
   TextField "OBJECT_28" at 588,256 size 72x32
   IOField "OBJECT_13" at 508,64 size 72x32
   IOField "OBJECT_14" at 508,112 size 72x32
   IOField "OBJECT_16" at 508,160 size 72x32
   IOField "OBJECT_18" at 508,256 size 72x32
   IOField "OBJECT_25" at 508,208 size 72x32
   IOField "OBJECT_27" at 508,304 size 72x32

screen "SetUpOperat1" 800x448, template "Template"
   TextField "OBJECT_3" at 80,144 size 216x32
   TextField "OBJECT_4" at 444,144 size 24x32
   TextField "OBJECT_8" at 444,208 size 24x32
   TextField "OBJECT_9" at 444,176 size 24x32
   TextField "OBJECT_10" at 444,240 size 24x32
   TextField "OBJECT_12" at 444,272 size 24x32
   TextField "OBJECT_14" at 444,304 size 24x32
   TextField "OBJECT_16" at 444,336 size 24x32
   TextField "OBJECT_17" at 268,88 size 104x32
   TextField "OBJECT_18" at 380,88 size 104x32
   TextField "OBJECT_19" at 380,112 size 104x32
   TextField "OBJECT_20" at 492,112 size 120x32
   TextField "OBJECT_21" at 492,88 size 120x32
   TextField "OBJECT_22" at 572,144 size 24x32
   TextField "OBJECT_23" at 572,208 size 24x32
   TextField "OBJECT_24" at 572,176 size 24x32
   TextField "OBJECT_25" at 572,240 size 24x32
   TextField "OBJECT_26" at 572,272 size 24x32
   TextField "OBJECT_27" at 572,304 size 24x32
   TextField "OBJECT_28" at 572,336 size 24x32
   TextField "OBJECT_31" at 572,368 size 24x32
   TextField "OBJECT_33" at 444,368 size 24x32
   TextField "OBJECT_74" at 156,32 size 504x32
   TextField "OBJECT_75" at 80,176 size 216x32
   TextField "OBJECT_76" at 80,208 size 216x32
   TextField "OBJECT_77" at 80,240 size 216x32
   TextField "OBJECT_78" at 80,272 size 216x32
   TextField "OBJECT_79" at 80,304 size 216x32
   TextField "OBJECT_80" at 80,336 size 216x32
   TextField "OBJECT_81" at 80,368 size 216x32
   SymbolicIOField "OBJECT_35" at 300,144 size 38x35
   IOField "OBJECT_36" at 380,144 size 56x32
   SymbolicIOField "OBJECT_37" at 300,240 size 38x35
   SymbolicIOField "OBJECT_38" at 300,208 size 38x35
   SymbolicIOField "OBJECT_39" at 300,176 size 38x35
   IOField "OBJECT_40" at 380,208 size 56x32
   IOField "OBJECT_41" at 380,176 size 56x32
   IOField "OBJECT_42" at 380,240 size 56x32
   SymbolicIOField "OBJECT_43" at 300,272 size 38x35
   IOField "OBJECT_44" at 380,272 size 56x32
   SymbolicIOField "OBJECT_45" at 300,304 size 38x35
   IOField "OBJECT_46" at 380,304 size 56x32
   SymbolicIOField "OBJECT_47" at 300,336 size 38x35
   IOField "OBJECT_48" at 380,336 size 56x32
   IOField "OBJECT_49" at 492,144 size 72x32
   IOField "OBJECT_50" at 492,176 size 72x32
   IOField "OBJECT_51" at 492,208 size 72x32
   IOField "OBJECT_52" at 492,240 size 72x32
   IOField "OBJECT_53" at 492,272 size 72x32
   IOField "OBJECT_54" at 492,304 size 72x32
   IOField "OBJECT_55" at 492,336 size 72x32
   SymbolicIOField "OBJECT_56" at 300,368 size 38x35
   IOField "OBJECT_58" at 492,368 size 72x32
   IOField "OBJECT_60" at 380,368 size 56x32
*)